//Station 3 - SMAC Homing Time Out
GVL_MASTER.stAlarms[3].aEventTimers[80]
(IN := (S_Master_SMAC.eState = E_SmacState.HOMING),PT:= T#30S );
IF GVL_MASTER.stAlarms[3].aEventTimers[80].Q  THEN 
	GVL_MASTER.stAlarms[3].aEventFlags[80] := TRUE;
END_IF
//Station 3 - SMAC Linear Homing fail
GVL_MASTER.stAlarms[3].aEventTimers[81]
(IN := (S_Master_SMAC.eState = E_SmacState.HOMING) AND stSmacIO.inStatusWordLinear.7 ,PT:= T#20S );
IF GVL_MASTER.stAlarms[3].aEventTimers[81].Q THEN 
	stAlarms[3].aEventFlags[81] := TRUE;
END_IF
//Station 3 - SMAC Linear Phasing fail
GVL_MASTER.stAlarms[3].aEventTimers[82]
(IN := (S_Master_SMAC.eState = E_SmacState.HOMING) AND stSmacIO.inStatusWordLinear.9 ,PT:= T#20S );
IF GVL_MASTER.stAlarms[3].aEventTimers[82].Q THEN
	stAlarms[3].aEventFlags[82] := TRUE;
END_IF
//Station 3 - SMAC Rotative Homing fail
GVL_MASTER.stAlarms[3].aEventTimers[83]
(IN := (S_Master_SMAC.eState = E_SmacState.HOMING) AND stSmacIO.inStatusWordRotative.7 ,PT:= T#20S );
IF GVL_MASTER.stAlarms[3].aEventTimers[83].Q THEN 
	stAlarms[3].aEventFlags[83] := TRUE;
END_IF
//Station 3 - SMAC Rotative Phasing fail
GVL_MASTER.stAlarms[3].aEventTimers[84]
(IN := (S_Master_SMAC.eState = E_SmacState.HOMING) AND stSmacIO.inStatusWordRotative.9 ,PT:= T#20S );
IF GVL_MASTER.stAlarms[3].aEventTimers[84].Q THEN 
	stAlarms[3].aEventFlags[84] := TRUE;
END_IF
END_ACTION

METHOD SetEventTexts : BOOL
VAR_INPUT
END_VAR
//Immediate Faults
GVL_MASTER.stAlarms[3].aEventTexts[1] := 'Station 3 - SMAC Linear General Fault';
GVL_MASTER.stAlarms[3].aEventTexts[2] := 'Station 3 - SMAC Linear Servo error';
GVL_MASTER.stAlarms[3].aEventTexts[3] := 'Station 3 - SMAC Rotative General Fault';
GVL_MASTER.stAlarms[3].aEventTexts[4] := 'Station 3 - SMAC Rotative Servo error';
GVL_MASTER.stAlarms[3].aEventTexts[5] := 'Station 3 - SMAC STO Fault';
GVL_MASTER.stAlarms[3].aEventTexts[6] := 'Station 3 - SMAC I2T Fault';
GVL_MASTER.stAlarms[3].aEventTexts[7] := 'Station 3 - SMAC Over temperature Fault';
GVL_MASTER.stAlarms[3].aEventTexts[8] := '';
GVL_MASTER.stAlarms[3].aEventTexts[9] := ''; 
GVL_MASTER.stAlarms[3].aEventTexts[10] := ''; 
GVL_MASTER.stAlarms[3].aEventTexts[11] := '';
GVL_MASTER.stAlarms[3].aEventTexts[12] := '';
GVL_MASTER.stAlarms[3].aEventTexts[13] := '';
GVL_MASTER.stAlarms[3].aEventTexts[14] := '';
GVL_MASTER.stAlarms[3].aEventTexts[15] := '';
GVL_MASTER.stAlarms[3].aEventTexts[16] := '';
GVL_MASTER.stAlarms[3].aEventTexts[17] := '';
GVL_MASTER.stAlarms[3].aEventTexts[18] := '';
GVL_MASTER.stAlarms[3].aEventTexts[19] := '';
GVL_MASTER.stAlarms[3].aEventTexts[20] := '';
GVL_MASTER.stAlarms[3].aEventTexts[21] := '';
GVL_MASTER.stAlarms[3].aEventTexts[22] := '';
GVL_MASTER.stAlarms[3].aEventTexts[28] := '';
GVL_MASTER.stAlarms[3].aEventTexts[29] := '';
GVL_MASTER.stAlarms[3].aEventTexts[30] := '';

//Cycle Stop Requests

GVL_MASTER.stAlarms[3].aEventTexts[80] := 'Station 3 - SMAC Homing Time Out';
GVL_MASTER.stAlarms[3].aEventTexts[81] := 'Station 3 - SMAC Linear Homing fail';
GVL_MASTER.stAlarms[3].aEventTexts[82] := 'Station 3 - SMAC Linear Phasing fail';
GVL_MASTER.stAlarms[3].aEventTexts[84] := 'Station 3 - SMAC Rotative Homing fail';
GVL_MASTER.stAlarms[3].aEventTexts[85] := 'Station 3 - SMAC Rotative Phasing fail';
GVL_MASTER.stAlarms[3].aEventTexts[86] := '';
GVL_MASTER.stAlarms[3].aEventTexts[87] := ''; 
GVL_MASTER.stAlarms[3].aEventTexts[88] := '';
GVL_MASTER.stAlarms[3].aEventTexts[89] := '';
END_METHOD

END_PROGRAM

// ---- POUs/00_MASTER/B_Safety.TcPOU
PROGRAM B_Safety
VAR


	bFirstRun						:BOOL:=TRUE;
	tonDelaySafetyRun				:Tc2_Standard.TON;
	
	
	bFirstSafetyErrorAck 			:BOOL;
	bSafetyErrorAck					:BOOL;	
	rTriggSafetyErrorAck  			:Tc2_Standard.R_TRIG;	
	tonDelayErrorAck				:Tc2_Standard.TON;
	tonSafetyErrorAckPulse			:Tc2_Standard.TON;


//-----------------------------------------------------oldschoo1
	
END_VAR

// Call for Actions:
a_Run_And_ErrorAck();
b_Cmd_SafetyDevices();
//----------------------oldschoo1

ACTION a_Run_And_ErrorAck:
// Run Safety PLC && ErrorAck: --------------------------------------------*
(**************************************************************************)


// Delay RUN on PowerUP
tonDelaySafetyRun(IN:=bFirstRun, 
				  PT:=tSystemPowerUP_Time);

IF tonDelaySafetyRun.Q 
	THEN
		GVL_MASTER.stSafety.bRunSafety 		:= TRUE;	
		bFirstRun 							:= FALSE;
		bFirstSafetyErrorAck 				:= TRUE;
END_IF

// Delay ErrorAck
tonDelayErrorAck(IN:=bFirstSafetyErrorAck, 
				 PT:=T#500MS);


// Trigger ErrorAck: ------------------------------------------------------*
rTriggSafetyErrorAck(CLK:=tonDelayErrorAck.Q OR 
						  bResetButtonRisingEdge);

IF rTriggSafetyErrorAck.Q 
	THEN
		bFirstSafetyErrorAck 	:= FALSE;
		bSafetyErrorAck 		:= TRUE;
END_IF


// Send Pulse for ErrorAck: -----------------------------------------------*
tonSafetyErrorAckPulse(IN:=bSafetyErrorAck, PT:=T#500MS);

IF bSafetyErrorAck 
							THEN
								GVL_MASTER.stSafety.bAckSafetyError := TRUE;
END_IF

IF tonSafetyErrorAckPulse.Q 
							THEN
								GVL_MASTER.stSafety.bAckSafetyError := FALSE;
								bSafetyErrorAck 					:= FALSE;
END_IF


//------------------------------------------------------------------oldschoo1
END_ACTION

ACTION b_Cmd_SafetyDevices:
// atm dev && test only 
	// map to:  stMachineStatus.bAutoCycle;  when done with dev/testing
	// map to:  stMachineStatus.bAutoCycle AND NOT stMachineStatus.bProcessCycle; //to allow operator to insert/take out the Pack fixture
  // map to:  stMachineStatus.bAutoCycle;  when done with dev/testing
IF stMachineStatus.bProcessCycle AND NOT Y_Master_Y_Axis.refY_Axis.Status.Moving THEN
	stSafety.bLightBeam_MuteCMD 	:= FALSE;
ELSE stSafety.bLightBeam_MuteCMD 	:= TRUE;
END_IF
	//stSafety.bLightBeam_MuteCMD 	:= TRUE;

IF stMachineStatus.bAutoCycle THEN
	stSafety.bTwoHands_MonitorCMD 	:= TRUE;
	stSafety.bLockDoor_CMD 			:= TRUE;
ELSE stSafety.bTwoHands_MonitorCMD 	:= FALSE;
	stSafety.bLockDoor_CMD 			:= FALSE;
END_IF
END_ACTION

ACTION z_HardwareHealth:
//to be finnished

(*
   	// TERMINAL 1 _ EK1100 - EtherCAT Coupler

	nEK1100State							AT %I*			:	UINT;	// Terminal INFO Data	
	sEK1100Status											:	STRING(200);
	

	// TERMINAL 2 _ EL6070-0033	- License Key Terminal for TC3
	
	nEL6070State							AT %I*			:	UINT;	// Terminal INFO Data	
	sEL6070Status											:	STRING(200);


	// TERMINAL 3 _ EL6910 - Safety PLC - Virtual Channels
	

	nEL6910State							AT %I*			:	UINT;	// Terminal INFO Data	
	sEL6910Status											:	STRING(200);


	// TERMINAL 4 _ EL1918 - 8 Channel Digital Safety Inputs
	

	nEL1918_1State							AT %I*			:	UINT;	// Terminal INFO Data	
	sEL1918Status											:	STRING(200);
	

	// TERMINAL 5 _ EL1918 - 8 Channel Digital Safety Inputs
                     	
	nEL1918_2State							AT %I*			:	UINT;	// Terminal INFO Data	
	sEL1918_2Status											:	STRING(200);
	

	// TERMINAL 6 _ ELEL2904 - 4 Channel Digital Safety Outputs


	nEL2904_1State							AT %I*			:	UINT;	// Terminal INFO Data	
	sEL2904_1Status											:	STRING(200);
	

	// TERMINAL 7 _ ELEL2904 - 4 Channel Digital Safety Outputs

		//Status* 
	nEL2904_2State							AT %I*			:	UINT;	// Terminal INFO Data	
	sEL2904_2Status											:	STRING(200);


	// TERMINAL 8 _ EL1809 - 16 Channel Digital Input Terminal
	
		//Status*	
	nEL1809_1State							AT %I*			:	UINT;	// Terminal INFO Data	
	sEL1809_1Status											:	STRING(200);
	
	iPSU_1_OK								AT %I*	 		: 	BOOL;	// Channel 03 - Power Supply Unit 1 OK
	iPSU_2_OK								AT %I*	 		: 	BOOL;	// Channel 04 - Power Supply Unit 2 OK
	iPSU_3_OK								AT %I*	 		: 	BOOL;	// Channel 05 - Power Supply Unit 3 OK	
	
	

	// TERMINAL 9 _ EL1809 - 16 Channel Digital Input Terminal

	nEL1809_2State							AT %I*			:	UINT;	// Terminal INFO Data
	sEL1809_2Status											:	STRING(200);
	
	// TERMINAL 10 _ EL2809	- 16 Channel Digital Output Terminal
	

	nEL2809State							AT %I*			:	UINT;	// Terminal INFO Data
	sEL2809Status											:	STRING(200);


	// TERMINAL 11 _ EL9576 - Brake Chopper Terminal

	nEL9576State							AT %I*			:	UINT;	// Terminal INFO Data
	sEL9576Status											:	STRING(200);
	

	// TERMINAL 12 _ EL7211-0010 - Servo Motor Drive

	nEL7211State							AT %I*			:	UINT;	// Terminal INFO Data
	sEL7211Status											:	STRING(200);	


	// BOX 13 _ maXYnos - Drive and Force Sensor

	nKistlermaXYmosState				   AT %I*		   :	UINT;	// Terminal INFO Data
	sKistlermaXYmosStatus								   :	STRING(200);	
	
	//--------------------------------------------------------------------------------------------------------------------------oldschoo1
*)
END_ACTION

END_PROGRAM

// ---- POUs/00_MASTER/C_Machine_CTRL.TcPOU
PROGRAM C_Machine_CTRL
VAR
	
	bFirstRun					:BOOL;
	bFirstAutoCycle				:BOOL;
	bSmacDone					:BOOL;
	bKistlerDone				:BOOL;
	rSmacDone					:R_TRIG;
	rKistlerDone				:R_TRIG;
	bStatisticsFlag				:ARRAY[0..1] OF BOOL;
	
	eMachineState				:E_MachineState:=E_MachineState.SYSTEM_POWER_UP;

	//Timers && Triggers
	tonSys_Init					:Tc2_Standard.TON:=(PT:=T#1S);
	tonSys_InitTimeout			:Tc2_Standard.TON:=(PT:=T#3M);					
	tonWAIT_SMAC_KISLR			:Tc2_Standard.TON;
	tonFirstAutoCycle			:Tc2_Standard.TON:=(PT:=T#500MS);
	
	//Process Cycle
	eCycleState					:E_ProcessCycle;
	stTotalReport				:ST_ProcessReport;
	bStartConditions			:BOOL;	
	tonTwoHandsTouching			:Tc2_Standard.TON;         
	bScrewPresent				: BOOL;
	bReservoirPresent			: BOOL;
	tonGrippersOpennedSignal	: TON;
	tonDelayExe					:Tc2_Standard.TON:=(PT:=T#100MS);
	rtrigResetModule			:Tc2_Standard.R_TRIG;
	rtrigProcessLogShift		:Tc2_Standard.R_TRIG;
	
	
	//Index
	idx							:INT;
	
END_VAR
//----------------------------------------------------------------------------oldschoo1

// Call for Actions

   b_Machine_Status();		//State machina 
	 c_ProcessCycle();	   //Master sequencer


//----------------------------------------------------------------*


// Process Report circular buffer
rtrigProcessLogShift(CLK:=eCycleState=E_ProcessCycle.Saving_DATA);

IF rtrigProcessLogShift.Q THEN 
	FOR idx:= 250 TO 2 BY -1 DO
		GVL_PERSISTENT.stProccessReportLog[idx]:=GVL_PERSISTENT.stProccessReportLog[idx-1];
	END_FOR
	GVL_PERSISTENT.stProccessReportLog[1]:=stTotalReport;
END_IF//																										||
//--------------------------------------------------------------------------------------------------------oldschoo1

ACTION b_Machine_Status:




//Timers && Triggers
tonSys_Init(IN:=stMachineStatus.bInitialising);
tonSys_InitTimeout(IN:=stMachineStatus.bInitialising);
IF stMachineStatus.eMachineState <> E_MachineState.SYSTEM_AUTO_CYCLE THEN
	bFirstAutoCycle							:= FALSE;
END_IF

//Transition IF Cycle Stop Fault OR Imediate Fault
IF NOT stMasterCtrl.bNoMachineImmediateFault THEN		
				stMachineStatus.eMachineState := E_MachineState.IMMEDIATE_FAULT;
	
ELSIF NOT stMasterCtrl.bNoCycleStopFault AND NOT stMachineStatus.bImmediateStopped THEN
				stMachineStatus.eMachineState := E_MachineState.CYCLE_STOP_FAULT;
END_IF

IF NOT GVL_Master.stMasterCTRL.bManualModeRequest THEN
	CMD_Axis.bManualMode	:=FALSE;
	CMD_Smac.bManualMode	:=FALSE;
	CMD_Kistler.bManualMode	:=FALSE;
END_IF
(****************************************************MACHINE_CTRL*******************************************************************)
//STATE MACHINE: ------------------------------------------------------------------------------------------------------------------SM
CASE stMachineStatus.eMachineState OF

E_MachineState.SYSTEM_POWER_UP: 		// ------------------------------------------------------------------------------POWER_UP

				IF tonSystemPowerUP.Q THEN
						stMachineStatus.eMachineState := E_MachineState.IMMEDIATE_STOPPED;//
				END_IF
	
E_MachineState.IMMEDIATE_STOPPED:		// ---------------------------------------------------------------------IMMEDIATE_STOPPED

				IF stMasterCtrl.bNoMachineImmediateFault AND bResetButtonFallingEdge THEN
						stMachineStatus.eMachineState := E_MachineState.SYSTEM_INITIALISING;//
						
				ELSIF NOT stMasterCtrl.bNoCycleStopFault THEN
						stMachineStatus.eMachineState := E_MachineState.CYCLE_STOP_FAULT;//
					
				ELSIF NOT stMasterCtrl.bNoMachineImmediateFault THEN
					stMachineStatus.eMachineState := E_MachineState.IMMEDIATE_FAULT;//	
				END_IF		


E_MachineState.SYSTEM_INITIALISING:		// -------------------------------------------------------------------SYSTEM_INITIALISING		

				IF tonSys_Init.Q THEN
						CMD_Axis.bEnable	:=TRUE;
						CMD_Smac.bEnable	:=TRUE;
						CMD_Kistler.bEnable	:=TRUE;
						
						CMD_Axis.bAbort		:=FALSE;
						CMD_Smac.bAbort		:=FALSE;
						CMD_Kistler.bAbort	:=FALSE;
				END_IF

				//IF Axis_STATUS.bReady AND Kistler_STATUS.bReady  AND Smac_STATUS.bReady THEN 
				 IF Axis_STATUS.bReady AND Kistler_STATUS.bReady AND ( GVL_PERSISTENT.bSMACEnable AND Smac_STATUS.bReady OR NOT GVL_PERSISTENT.bSMACEnable) THEN //**LAA  29092025
										stMachineStatus.eMachineState:= E_MachineState.SYSTEM_READY_TO_START;//
				END_IF

				IF bStopButtonFallingEdge OR 
			 	  (stMasterCtrl.bNoMachineImmediateFault AND 
			 	  (stMasterCtrl.bCycleStopRequest OR tonSys_InitTimeout.Q) AND 
			       stMasterCtrl.bAllActionsStopped)
					THEN
										stMachineStatus.eMachineState := E_MachineState.CYCLE_STOPPED;//
						
				ELSIF stMasterCtrl.bNoMachineImmediateFault AND NOT stMasterCtrl.bNoCycleStopFault 
					THEN		
										stMachineStatus.eMachineState := E_MachineState.CYCLE_STOP_FAULT;//
			
				ELSIF NOT stMasterCtrl.bNoMachineImmediateFault 
					THEN
										stMachineStatus.eMachineState := E_MachineState.IMMEDIATE_FAULT;//
				END_IF
			
					
E_MachineState.SYSTEM_READY_TO_START:	// -------------------------------------------------------------------SYSTEM_READY_TO_START<<<

				IF 	 bStartButtonFallingEdge AND stMasterCtrl.bAllModulesReady THEN
					
										stMachineStatus.eMachineState := E_MachineState.SYSTEM_AUTO_CYCLE;//
				
				ELSIF bStopButtonFallingEdge THEN
					
										stMachineStatus.eMachineState := E_MachineState.STOPPING;//
										
				ELSIF stMasterCtrl.bNoMachineImmediateFault AND NOT stMasterCtrl.bNoCycleStopFault THEN	
	
										stMachineStatus.eMachineState := E_MachineState.CYCLE_STOP_FAULT;//
			
				ELSIF NOT stMasterCtrl.bNoMachineImmediateFault THEN
										stMachineStatus.eMachineState := E_MachineState.IMMEDIATE_FAULT;//
				ELSIF GVL_Master.stMasterCTRL.bManualModeRequest AND stMasterCtrl.bNoMachineImmediateFault AND stMasterCtrl.bNoCycleStopFault THEN
										stMachineStatus.eMachineState := E_MachineState.MANUAL_MODE;//
				END_IF

				

E_MachineState.SYSTEM_AUTO_CYCLE:		// ---------------------------------------------------------------------SYSTEM_AUTO_CYCLE	

				IF bStopButtonFallingEdge THEN					
										stMachineStatus.eMachineState := E_MachineState.STOPPING;//
						
				ELSIF stMasterCtrl.bCycleStopRequest THEN 
					
										stMachineStatus.eMachineState := E_MachineState.STOPPING;//
										
				ELSIF stMasterCtrl.bNoMachineImmediateFault AND NOT stMasterCtrl.bNoCycleStopFault THEN	
	
										stMachineStatus.eMachineState := E_MachineState.CYCLE_STOP_FAULT;//
			
				ELSIF NOT stMasterCtrl.bNoMachineImmediateFault THEN
										stMachineStatus.eMachineState := E_MachineState.IMMEDIATE_FAULT;//
				END_IF	

E_MachineState.SYSTEM_STANDBY:;//



E_MachineState.STOPPING:				// ------------------------------------------------------------------------------STOPPING

				IF stMasterCtrl.bAllActionsStopped THEN
										stMachineStatus.eMachineState := E_MachineState.CYCLE_STOPPED;//					
				END_IF
				CMD_Axis.bEnable	:=FALSE;
				CMD_Smac.bEnable	:=FALSE;
				CMD_Kistler.bEnable	:=FALSE;
				
				CMD_Axis.bAbort		:=TRUE;
				CMD_Smac.bAbort		:=TRUE;
				CMD_Kistler.bAbort	:=TRUE;

E_MachineState.CYCLE_STOPPED:			// -------------------------------------------------------------------------CYCLE_STOPPED

				IF stMasterCtrl.bNoCycleStopFault   AND 
	      		NOT stMasterCtrl.bCycleStopRequest  AND 
                               bResetButtonFallingEdge

									THEN	
										stMachineStatus.eMachineState := E_MachineState.SYSTEM_INITIALISING;		
				END_IF	

E_MachineState.IMMEDIATE_FAULT:			// -----------------------------------------------------------------------IMMEDIATE_FAULT
				
				CMD_Axis.bEnable	:=FALSE;
				CMD_Smac.bEnable	:=FALSE;
				CMD_Kistler.bEnable	:=FALSE;
						
				CMD_Axis.bAbort		:=TRUE;
				CMD_Smac.bAbort		:=TRUE;
				CMD_Kistler.bAbort	:=TRUE;
				
				IF stMasterCtrl.bNoMachineImmediateFault	THEN
										stMachineStatus.eMachineState := E_MachineState.IMMEDIATE_STOPPED;		
				END_IF

E_MachineState.CYCLE_STOP_FAULT:		// ----------------------------------------------------------------------CYCLE_STOP_FAULT

				CMD_Axis.bEnable	:=FALSE;
				CMD_Smac.bEnable	:=FALSE;
				CMD_Kistler.bEnable	:=FALSE;
						
				CMD_Axis.bAbort		:=TRUE;
				CMD_Smac.bAbort		:=TRUE;
				CMD_Kistler.bAbort	:=TRUE;
				
				IF stMasterCtrl.bNoCycleStopFault THEN
										stMachineStatus.eMachineState := E_MachineState.CYCLE_STOPPED;
				END_IF	


E_MachineState.MANUAL_MODE:;//

				IF bStopButtonFallingEdge OR NOT GVL_Master.stMasterCTRL.bManualModeRequest THEN
					
										stMachineStatus.eMachineState := E_MachineState.STOPPING;//
										
										CMD_Axis.bManualMode:=FALSE;
										CMD_Smac.bManualMode:=FALSE;
										CMD_Kistler.bManualMode:=FALSE;
										CMD_Axis.bAbort		:=TRUE;
										CMD_Smac.bAbort		:=TRUE;
										CMD_Kistler.bAbort	:=TRUE;
				ELSIF stMasterCtrl.bNoMachineImmediateFault AND NOT stMasterCtrl.bNoCycleStopFault THEN	
	
										stMachineStatus.eMachineState := E_MachineState.CYCLE_STOP_FAULT;//
										
										CMD_Axis.bManualMode:=FALSE;
										CMD_Smac.bManualMode:=FALSE;
										CMD_Kistler.bManualMode:=FALSE;
										CMD_Axis.bAbort		:=TRUE;
										CMD_Smac.bAbort		:=TRUE;
										CMD_Kistler.bAbort	:=TRUE;
			
				ELSIF NOT stMasterCtrl.bNoMachineImmediateFault THEN
							
										stMachineStatus.eMachineState := E_MachineState.IMMEDIATE_FAULT;//
				
										CMD_Axis.bManualMode:=FALSE;
										CMD_Smac.bManualMode:=FALSE;
										CMD_Kistler.bManualMode:=FALSE;
										CMD_Axis.bAbort		:=TRUE;
										CMD_Smac.bAbort		:=TRUE;
										CMD_Kistler.bAbort	:=TRUE;
										
				ELSE 					CMD_Axis.bManualMode:=TRUE;
										CMD_Smac.bManualMode:=TRUE;
										CMD_Kistler.bManualMode:=TRUE;
				END_IF
ELSE
stMachineStatus.eMachineState:=E_MachineState.SYSTEM_POWER_UP;		
END_CASE									// ------------------------------------------------------------------------------- END SM


(******************************************************MACHINE_STATUS***************************************************************)
// Status Flags -----------------------------------------------------------------------------------------------------STATUS_FLAGS
stMachineStatus.bSystemPowerUp 			:= (stMachineStatus.eMachineState = E_MachineState.SYSTEM_POWER_UP);
stMachineStatus.bImmediateStopped 		:= (stMachineStatus.eMachineState = E_MachineState.IMMEDIATE_STOPPED);
stMachineStatus.bInitialising 			:= (stMachineStatus.eMachineState = E_MachineState.SYSTEM_INITIALISING);
stMachineStatus.bReadyToStart 			:= (stMachineStatus.eMachineState = E_MachineState.SYSTEM_READY_TO_START);
stMachineStatus.bAutoCycle 				:= (stMachineStatus.eMachineState = E_MachineState.SYSTEM_AUTO_CYCLE);
stMachineStatus.bStandby 				:= (stMachineStatus.eMachineState = E_MachineState.SYSTEM_STANDBY);
stMachineStatus.bStopping 				:= (stMachineStatus.eMachineState = E_MachineState.STOPPING);
stMachineStatus.bCycleStopped 			:= (stMachineStatus.eMachineState = E_MachineState.CYCLE_STOPPED);
stMachineStatus.bImmediateFault 		:= (stMachineStatus.eMachineState = E_MachineState.IMMEDIATE_FAULT);
stMachineStatus.bCycleStopFault 		:= (stMachineStatus.eMachineState = E_MachineState.CYCLE_STOP_FAULT);
stMachineStatus.bManualMode 			:= (stMachineStatus.eMachineState = E_MachineState.MANUAL_MODE);

//Transition Flags -----------------------------------------------------------------------------------------------TRANZITION_FLAGS
stMasterCtrl.bAllActionsStopped			:= (Axis_STATUS.bReady AND Kistler_STATUS.bReady AND ( GVL_PERSISTENT.bSMACEnable AND Smac_STATUS.bReady OR NOT GVL_PERSISTENT.bSMACEnable) ) OR  //**LAA 29092025
										   (NOT Axis_STATUS.bBusy AND NOT Kistler_STATUS.bBusy );
										   
stMasterCtrl.bAllModulesReady			:= (Axis_STATUS.bReady AND Kistler_STATUS.bReady AND ( GVL_PERSISTENT.bSMACEnable AND Smac_STATUS.bReady OR NOT GVL_PERSISTENT.bSMACEnable)); //**LAA 29092025

(*stMasterCtrl.bAllActionsStopped			:= (Axis_STATUS.bReady AND Kistler_STATUS.bReady AND Smac_STATUS.bReady ) OR
										   (NOT Axis_STATUS.bBusy AND NOT Kistler_STATUS.bBusy );
										   
stMasterCtrl.bAllModulesReady			:= (Axis_STATUS.bReady AND Kistler_STATUS.bReady AND Smac_STATUS.bReady ); 

*)
END_ACTION

ACTION c_ProcessCycle:
//Timers
tonDelayExe(IN:=(eCycleState=E_ProcessCycle.AXIS_HOME AND Axis_STATUS.bReady) OR
				(eCycleState=E_ProcessCycle.AXIS_CMD_1 AND Axis_STATUS.bReady) OR
				(eCycleState=E_ProcessCycle.AXIS_CMD_2 AND Axis_STATUS.bReady) OR
				(eCycleState=E_ProcessCycle.AXIS_CMD_3 AND Axis_STATUS.bReady) OR
				(eCycleState=E_ProcessCycle.SMAC_CMD_1 AND Smac_STATUS.bReady) OR
				((eCycleState=E_ProcessCycle.CMD_SMAC_KISLR OR eCycleState=E_ProcessCycle.CMD_KISLR )AND (CMD_Kistler.bExecute OR NOT bReservoir_Present)AND (GVL_PERSISTENT.bSMACEnable AND CMD_Smac.bExecute OR NOT bScrewPresent ))
);  //AND Smac_STATUS.bReady));				//to finish
				
tonGrippersOpennedSignal( IN :=  NOT stSmac.bGripperA_ClosedSensor AND NOT stSmac.bGripperA_ClosedSensor, PT := T#1S);
tonWAIT_SMAC_KISLR(IN := eCycleState = E_ProcessCycle.WAIT_SMAC_KISLR,PT := T#500MS);
tonFirstAutoCycle( IN := eCycleState = E_ProcessCycle.IDLE AND stMachineStatus.bAutoCycle);
(******************************************************START CONDITIONS******************************************************)				
// Start Conditions: 
// - Optional add HMI PopUp if Pack fixture is in but NOT all 3 parts present -	
		
tonTwoHandsTouching(IN:=stSafety.bTwoHands_Signal, PT:=T#500MS);       // **LAA 03/12/2025 > it was too slow PT:=T#2S);

bStartConditions 		 := (tonTwoHandsTouching.Q AND 
							stMachineStatus.bAutoCycle AND
							GVL_MASTER.bPuck_Present);
							//AND bGearBox_Present 
					
							
//Reset Module --------------------------------------------------------------------------------------------------------------*
IF bResetButtonRisingEdge OR 
stMachineStatus.bCycleStopFault OR stMachineStatus.bImmediateFault OR stMachineStatus.bImmediateStopped
THEN eCycleState:=E_ProcessCycle.RESET_ALL_CMD;END_IF
//KISTLER / SMAC DONE---------------------------------------------------------------------------------------------------------*
rSmacDone( CLK := Smac_STATUS.bDone );					
rKistlerDone( CLK := Kistler_STATUS.bDone );					

IF rKistlerDone.Q THEN 
	bKistlerDone		:= TRUE;
END_IF
IF rSmacDone.Q THEN
	bSmacDone			:= TRUE;
END_IF

(************************************************************CTRL*************************************************************)
//STATE MACHINE: -----------------------------------------------------------------------------------------------------------SM
CASE eCycleState OF
						(****************************************************************IDLE********************************)
E_ProcessCycle.IDLE:	//-----------------------------------------------------------------------------------------------IDLE
									IF bStartConditions AND GVL_PERSISTENT.bSMACEnable THEN   //**LAA 29092025
										eCycleState:=E_ProcessCycle.AXIS_CMD_1;
										stTotalReport.bKis_Pass								:= FALSE;
										stTotalReport.bKis_Fail								:= FALSE;
										stTotalReport.bSmac_Pass							:= FALSE;
										stTotalReport.bSmac_Fail							:= FALSE;
										GVL_IO.qCycleIndicator_RedLED						:= FALSE;
										GVL_IO.qCycleIndicator_GreenLED						:= FALSE;
										S_Master_SMAC.bCloseGripper							:= FALSE;
										ELSIF bStartConditions AND NOT GVL_PERSISTENT.bSMACEnable THEN // *LAA  29092025
											eCycleState:=E_ProcessCycle.AXIS_CMD_2;
											stTotalReport.bKis_Pass								:= FALSE;
											stTotalReport.bKis_Fail								:= FALSE;
											stTotalReport.bSmac_Pass							:= FALSE;
											stTotalReport.bSmac_Fail							:= FALSE;
											GVL_IO.qCycleIndicator_RedLED						:= FALSE;
											GVL_IO.qCycleIndicator_GreenLED						:= FALSE;
											S_Master_SMAC.bCloseGripper							:= FALSE;
									END_IF
									 IF NOT bFirstAutoCycle AND GVL_MASTER.bPuck_Present AND
										NOT tonFirstAutoCycle.Q AND stMachineStatus.bAutoCycle THEN
										eCycleState:=E_ProcessCycle.AXIS_CMD_3;
										stTotalReport.bKis_Pass								:= FALSE;
										stTotalReport.bKis_Fail								:= FALSE;
										stTotalReport.bSmac_Pass							:= FALSE;
										stTotalReport.bSmac_Fail							:= FALSE;
										GVL_IO.qCycleIndicator_RedLED						:= FALSE;
										GVL_IO.qCycleIndicator_GreenLED						:= FALSE;
										S_Master_SMAC.bCloseGripper							:= FALSE;
									END_IF
									//Just Idleing like chilling here
									CMD_Smac.bFixtureGripper		:= FALSE;
									CMD_Smac.bGuideGripper			:= FALSE;
									IF stMachineStatus.bAutoCycle AND NOT GVL_MASTER.bPuck_Present THEN
										GVL_HMI.sMessageToOperator	:='Insert Nest';
									ELSIF stMachineStatus.bAutoCycle AND GVL_MASTER.bPuck_Present THEN
										GVL_HMI.sMessageToOperator	:='Put two hands to start Cycle Process';
									ELSIF NOT stMachineStatus.bAutoCycle AND  stMachineStatus.bReadyToStart THEN
									GVL_HMI.sMessageToOperator	:='Press START to Begin';
									ELSIF NOT stMachineStatus.bAutoCycle AND  NOT stMachineStatus.bReadyToStart THEN
									GVL_HMI.sMessageToOperator	:='Press RESET';
									END_IF
									
							(************************************************************CYCLE******************************)									
E_ProcessCycle.AXIS_CMD_1:	//-------------------------------------------------------------------------------------AXIS_CMD_1

									IF Axis_STATUS.bReady THEN
											stY_Axis.bSetToPosition[1]	:=TRUE;
									END_IF

									IF tonDelayExe.Q THEN
											CMD_Axis.bExecute			:=TRUE;
											eCycleState:=E_ProcessCycle.WAIT_AXIS_CMD_1;
									END_IF
									GVL_HMI.sMessageToOperator	:='Axis Y Moving to Position 1';
									bFirstAutoCycle						:=TRUE;
									
	
E_ProcessCycle.WAIT_AXIS_CMD_1:	//----------------------------------------------------------------------------WAIT_AXIS_CMD_1
							 		IF GVL_PERSISTENT.bSMACEnable AND Axis_STATUS.bDone AND bScrew_Present THEN
											stY_Axis.bSetToPosition[1]	:=FALSE;
											CMD_Axis.bExecute			:=FALSE;
											bScrewPresent				:=TRUE;
											eCycleState:=E_ProcessCycle.SMAC_CMD_1;
									ELSIF  GVL_PERSISTENT.bSMACEnable AND Axis_STATUS.bDone AND NOT bScrew_Present OR NOT GVL_PERSISTENT.bSMACEnable THEN
											stY_Axis.bSetToPosition[1]	:=FALSE;
											CMD_Axis.bExecute			:=FALSE;
											bScrewPresent				:=FALSE;
											eCycleState:=E_ProcessCycle.AXIS_CMD_2;
									END_IF
									
									
E_ProcessCycle.SMAC_CMD_1:	//-------------------------------------------------------------------------------------SMAC_CMD_1		//to finish
									IF  Smac_STATUS.bReady THEN
										stSmac.bSet_PickScrew				:=TRUE;
										CMD_Smac.bExecute					:=TRUE;
									END_IF
									IF  Smac_Status.bBusy THEN
										eCycleState:=E_ProcessCycle.WAIT_SMAC_CMD_1;
									END_IF
									
									GVL_HMI.sMessageToOperator	:='Smac Picking Screw Part';

	
E_ProcessCycle.WAIT_SMAC_CMD_1:	//----------------------------------------------------------------------------WAIT_SMAC_CMD_1		//to finish
									//Wait for Smac device to feedback 
									IF Smac_STATUS.bFirstPartOfCycleDone THEN
										eCycleState:=E_ProcessCycle.AXIS_CMD_2;	
										CMD_Smac.bExecute				:=FALSE;
									END_IF

E_ProcessCycle.AXIS_CMD_2:	//-------------------------------------------------------------------------------------AXIS_CMD_2
							 		
											stY_Axis.bSetToPosition[2]	:=TRUE;
									

									IF tonDelayExe.Q AND Axis_STATUS.bReady THEN
											CMD_Axis.bExecute			:=TRUE;
											eCycleState:=E_ProcessCycle.WAIT_AXIS_CMD_2;
									END_IF	
									
									GVL_HMI.sMessageToOperator	:='Axis Y Moving to Position 2';

E_ProcessCycle.WAIT_AXIS_CMD_2:	//----------------------------------------------------------------------------WAIT_AXIS_CMD_2
						 		IF Axis_STATUS.bDone  AND GVL_PERSISTENT.bSMACEnable THEN
											stY_Axis.bSetToPosition[2]	:=FALSE;
											CMD_Axis.bExecute			:=FALSE;
											eCycleState:=E_ProcessCycle.GRIPPERS_CMD_1;
											ELSIF Axis_STATUS.bDone AND NOT GVL_PERSISTENT.bSMACEnable THEN 
												stY_Axis.bSetToPosition[2]	:=FALSE;
												CMD_Axis.bExecute			:=FALSE;
												eCycleState:=E_ProcessCycle.CMD_KISLR;;
									END_IF	
E_ProcessCycle.GRIPPERS_CMD_1: //------------------------------------------------------------------------------GRIPPERS_CMD_1
								
									CMD_Smac.bFixtureGripper		:= TRUE;
									CMD_Smac.bGuideGripper			:= TRUE;
								
								eCycleState:=E_ProcessCycle.WAIT_GRIPPERS_CMD_1;
								
								

E_ProcessCycle.WAIT_GRIPPERS_CMD_1: //--------------------------------------------------------------------WAIT_GRIPPERS_CMD_1
								IF stSmac.bGripperA_ClosedSensor AND stSmac.bGripperA_ClosedSensor AND 
									(bScrewPresent OR bPuck_Present) THEN
									eCycleState:=E_ProcessCycle.CMD_SMAC_KISLR;
								ELSIF stSmac.bGripperA_ClosedSensor AND stSmac.bGripperA_ClosedSensor AND // *LAA ????????
									(bScrewPresent OR bPuck_Present) THEN
									eCycleState:=E_ProcessCycle.STORE_PROC_DATA;
								END_IF

E_ProcessCycle.CMD_SMAC_KISLR:	//-------------------------------------------------------------------------CMD_SMAC_AND_KISLR		//to finish
							 		IF Kistler_STATUS.bReady THEN // AND Smac_STATUS.bReady
											IF bReservoir_Present THEN
												CMD_Kistler.bExecute		:=TRUE;
												bReservoirPresent			:=TRUE;
											END_IF
											IF bScrewPresent THEN
											stSmac.bSet_ScrewItIn		:=TRUE;
											CMD_Smac.bExecute			:=TRUE;
											END_IF
									END_IF

									IF tonDelayExe.Q THEN
										
											eCycleState:=E_ProcessCycle.WAIT_SMAC_KISLR;
									END_IF				
									GVL_HMI.sMessageToOperator	:='Kistler and Screw Process';

E_ProcessCycle.WAIT_SMAC_KISLR:	//----------------------------------------------------------------------------WAIT_SMAC_KISLR		//to finish
						 			IF (bKistlerDone OR NOT bReservoir_Present) AND (bSmacDone OR NOT bScrewPresent) THEN
											CMD_Kistler.bExecute		:=FALSE;
											stSmac.bSet_ScrewItIn		:=FALSE;
											CMD_Smac.bExecute			:=FALSE;
											//open guide gripper
											eCycleState:=E_ProcessCycle.STORE_PROC_DATA;
									END_IF	
//**************************************LAA******************************************************************//			

E_ProcessCycle.CMD_KISLR:	//-------------------------------------------------------------------------CMD_SMAC_AND_KISLR		//to finish
							 		IF Kistler_STATUS.bReady THEN // AND Smac_STATUS.bReady
											IF bReservoir_Present THEN
												CMD_Kistler.bExecute		:=TRUE;
												bReservoirPresent			:=TRUE;
											END_IF
									END_IF

									IF tonDelayExe.Q THEN
										
											eCycleState:=E_ProcessCycle.WAIT_KISLR;
									END_IF				
									GVL_HMI.sMessageToOperator	:='Kistler processing';

E_ProcessCycle.WAIT_KISLR:	//----------------------------------------------------------------------------WAIT_SMAC_KISLR		//to finish
						 			IF (bKistlerDone OR NOT bReservoir_Present) THEN
											CMD_Kistler.bExecute		:=FALSE;
											eCycleState:=E_ProcessCycle.STORE_PROC_DATA;
									END_IF	
//**************************************LAA******************************************************************//			
E_ProcessCycle.STORE_PROC_DATA:	//----------------------------------------------------------------------------STORE_PROC_DATA		//to finish
		
	bKistlerDone 			:= FALSE;
	bSmacDone 				:= FALSE;
	
	IF bReservoirPresent THEN
		stTotalReport.bKis_Pass								:=K_Master_Kistler.stKistlerReport.bKis_Pass;
		stTotalReport.bKis_Fail								:=K_Master_Kistler.stKistlerReport.bKis_Fail;
		stTotalReport.rKis_HighestRecordedForce				:=K_Master_Kistler.stKistlerReport.rKis_HighestRecordedForce;
		stTotalReport.rKis_LowestRecordedForce				:=K_Master_Kistler.stKistlerReport.rKis_LowestRecordedForce;
		stTotalReport.rKis_DistanceRecord					:=K_Master_Kistler.stKistlerReport.rKis_DistanceRecord;
		stTotalReport.rKis_Settings_ForceUpperTreshold		:=K_Master_Kistler.stKistlerReport.rKis_Settings_ForceUpperTreshold;
		stTotalReport.rKis_Settings_ForceLowerTreshold		:=K_Master_Kistler.stKistlerReport.rKis_Settings_ForceLowerTreshold;
		stTotalReport.rKis_Settings_StartMeasurePoint		:=K_Master_Kistler.stKistlerReport.rKis_Settings_StartMeasurePoint;
		stTotalReport.rKis_Settings_ReservoirBottomPoint	:=K_Master_Kistler.stKistlerReport.rKis_Settings_ReservoirBottomPoint;
		IF stTotalReport.bKis_Pass THEN
			stTotalReport.sKis_Result							:='PASS';
		ELSIF stTotalReport.bKis_FaiL THEN
			stTotalReport.sKis_Result							:='FAIL';
		ELSE stTotalReport.sKis_Result							:='';
		END_IF
	ELSE
		stTotalReport.bKis_Pass								:=FALSE;
		stTotalReport.bKis_Fail								:=FALSE;
		stTotalReport.rKis_HighestRecordedForce				:=0;
		stTotalReport.rKis_LowestRecordedForce				:=0;
		stTotalReport.rKis_Settings_ForceUpperTreshold		:=0;
		stTotalReport.rKis_Settings_ForceLowerTreshold		:=0;
		stTotalReport.rKis_Settings_StartMeasurePoint		:=0;
		stTotalReport.rKis_Settings_ReservoirBottomPoint	:=0;
		stTotalReport.sKis_Result							:='';
	END_IF
	IF GVL_PERSISTENT.bSMACEnable AND bScrewPresent THEN
		stTotalReport.rSmac_Settings_LinearAcc				:=S_Master_SMAC.stSmacReport.rSmac_Settings_LinearAcc;
		stTotalReport.rSmac_Settings_LinearVel				:=S_Master_SMAC.stSmacReport.rSmac_Settings_LinearVel;
		stTotalReport.rSmac_Settings_RotativeAcc			:=S_Master_SMAC.stSmacReport.rSmac_Settings_RotativeAcc;
		stTotalReport.rSmac_Settings_RotativeVel			:=S_Master_SMAC.stSmacReport.rSmac_Settings_RotativeVel;
		stTotalReport.rSmac_Settings_LinearTorque			:=S_Master_SMAC.stSmacReport.rSmac_Settings_LinearTorque;
		stTotalReport.rSmac_MaxDistanceReached				:=S_Master_SMAC.stSmacReport.rSmac_MaxDistanceReached;
		stTotalReport.bSmac_Pass							:=S_Master_SMAC.stSmacReport.bSmac_Pass;
		stTotalReport.bSmac_Fail							:=S_Master_SMAC.stSmacReport.bSmac_Fail;
		IF stTotalReport.bSmac_Pass THEN
			stTotalReport.sSmac_Result							:='PASS';
		ELSIF stTotalReport.bSmac_Fail THEN
			stTotalReport.sSmac_Result							:='FAIL';
		ELSE stTotalReport.sSmac_Result							:='';
		END_IF
	ELSE
		stTotalReport.rSmac_Settings_LinearAcc				:=0;
		stTotalReport.rSmac_Settings_LinearVel				:=0;
		stTotalReport.rSmac_Settings_RotativeAcc			:=0;
		stTotalReport.rSmac_Settings_RotativeVel			:=0;
		stTotalReport.rSmac_Settings_LinearTorque			:=0;
		stTotalReport.rSmac_MaxDistanceReached				:=0;
		stTotalReport.bSmac_Pass							:=FALSE;
		stTotalReport.bSmac_Fail							:=FALSE;
		stTotalReport.sSmac_Result							:='';
	END_IF
	
	stTotalReport.sDate										:= GVL_MASTER.sSystemDate;
	stTotalReport.sTime										:= GVL_MASTER.sSystemTime;
	
	//STATISTICS
	IF bReservoirPresent AND stTotalReport.bKis_Pass AND NOT bStatisticsFlag[0] THEN
		GVL_PERSISTENT.nKistlerGoodParts					:= GVL_PERSISTENT.nKistlerGoodParts + 1;
		GVL_PERSISTENT.nKistlerTotalGoodParts				:= GVL_PERSISTENT.nKistlerTotalGoodParts + 1;
		bStatisticsFlag[0]									:= TRUE;
	END_IF
	IF bReservoirPresent AND stTotalReport.bKis_Fail AND NOT bStatisticsFlag[0] THEN
		GVL_PERSISTENT.nKistlerBadParts						:= GVL_PERSISTENT.nKistlerBadParts + 1;
		GVL_PERSISTENT.nKistlerTotalBadParts				:= GVL_PERSISTENT.nKistlerTotalBadParts + 1;
		bStatisticsFlag[0]									:= TRUE;
	END_IF
	
	IF bScrewPresent AND stTotalReport.bSmac_Pass AND NOT bStatisticsFlag[1] THEN
		GVL_PERSISTENT.nSmacGoodParts						:= GVL_PERSISTENT.nSmacGoodParts + 1;
		GVL_PERSISTENT.nSmacTotalGoodParts					:= GVL_PERSISTENT.nSmacTotalGoodParts + 1;
		bStatisticsFlag[1]									:= TRUE;
	END_IF
		IF bScrewPresent AND stTotalReport.bSmac_Fail AND NOT bStatisticsFlag[1] THEN
		GVL_PERSISTENT.nSmacBadParts						:= GVL_PERSISTENT.nSmacBadParts + 1;
		GVL_PERSISTENT.nSmacTotalBadParts					:= GVL_PERSISTENT.nSmacTotalBadParts + 1;
		bStatisticsFlag[1]									:= TRUE;
	END_IF
	
			
			
									eCycleState:=E_ProcessCycle.Saving_DATA;	
E_ProcessCycle.Saving_DATA: //------------------------------------------------------------------------------------Saving_DATA
									eCycleState:=E_ProcessCycle.GRIPPERS_CMD_2;
									bStatisticsFlag[0]									:= FALSE;
									bStatisticsFlag[1]									:= FALSE;
									IF (bReservoirPresent AND stTotalReport.bKis_Pass) OR 
										(bScrewPresent AND stTotalReport.bSmac_Pass)THEN
										GVL_IO.qCycleIndicator_GreenLED						:= TRUE;
									ELSIF (bReservoirPresent AND stTotalReport.bKis_Fail) OR 
										(bScrewPresent AND stTotalReport.bSmac_Fail) THEN
										GVL_IO.qCycleIndicator_RedLED						:= TRUE;		
									END_IF
E_ProcessCycle.GRIPPERS_CMD_2: //------------------------------------------------------------------------------GRIPPERS_CMD_1
								
								CMD_Smac.bFixtureGripper		:= FALSE;
								CMD_Smac.bGuideGripper			:= FALSE;
								
								eCycleState:=E_ProcessCycle.WAIT_GRIPPERS_CMD_2;
								
								
								

E_ProcessCycle.WAIT_GRIPPERS_CMD_2: //--------------------------------------------------------------------WAIT_GRIPPERS_CMD_1
								IF tonGrippersOpennedSignal.Q THEN
								eCycleState:=E_ProcessCycle.AXIS_CMD_3;
								END_IF
			
E_ProcessCycle.AXIS_CMD_3:	//-------------------------------------------------------------------------------------AXIS_CMD_3
						 		IF Axis_STATUS.bReady THEN
											stY_Axis.bSetToPosition[3]	:=TRUE;
									END_IF

									IF tonDelayExe.Q THEN
											CMD_Axis.bExecute			:=TRUE;
											eCycleState:=E_ProcessCycle.WAIT_AXIS_CMD_3;
									END_IF		
								GVL_HMI.sMessageToOperator	:='Take Nest please';

E_ProcessCycle.WAIT_AXIS_CMD_3:	//----------------------------------------------------------------------------WAIT_AXIS_CMD_3
							 		IF Axis_STATUS.bDone THEN
											stY_Axis.bSetToPosition[3]	:=FALSE;
											CMD_Axis.bExecute			:=FALSE;
											eCycleState:=E_ProcessCycle.AXIS_HOME;
									END_IF


E_ProcessCycle.AXIS_HOME:	//-------------------------------------------------------------------------------------AXIS_HOME
							 		IF Axis_STATUS.bReady THEN
											stY_Axis.bSetToHome			:=TRUE;
											Y_Master_Y_Axis.bRetract 	:=TRUE;
									END_IF

									IF tonDelayExe.Q THEN
											CMD_Axis.bExecute			:=TRUE;
											eCycleState:=E_ProcessCycle.WAIT_AXIS_HOME;
									END_IF
									GVL_HMI.sMessageToOperator	:='Axis Y Homing';

E_ProcessCycle.WAIT_AXIS_HOME:	//----------------------------------------------------------------------------WAIT_AXIS_HOME
							 		IF Axis_STATUS.bDone THEN
											stY_Axis.bSetToHome			:=FALSE;
											CMD_Axis.bExecute			:=FALSE;
											Y_Master_Y_Axis.bRetract 	:=FALSE;
											eCycleState:=E_ProcessCycle.IDLE;
									END_IF
									bFirstAutoCycle						:=TRUE;

									
								(*********************************************************RESET*****************************)
E_ProcessCycle.RESET_ALL_CMD:	//------------------------------------------------------------------------------RESET_ALL_CMD

											CMD_Axis.bExecute									:=FALSE;
											CMD_Smac.bExecute									:=FALSE;
											CMD_Kistler.bExecute								:=FALSE;
											
											stSmac.bSet_PickScrew								:=FALSE;											
											stSmac.bSet_ScrewItIn								:=FALSE;
											CMD_Smac.bFixtureGripper							:= FALSE;
											CMD_Smac.bGuideGripper								:= FALSE;


											stY_Axis.bSetToHome									:=FALSE;
											Y_Master_Y_Axis.bRetract 							:=FALSE;
											stY_Axis.bSetToPosition[1]							:=FALSE;
											stY_Axis.bSetToPosition[2]							:=FALSE;
											stY_Axis.bSetToPosition[3]							:=FALSE;
											
											bKistlerDone 										:= FALSE;
											bSmacDone 											:= FALSE;
											bScrewPresent										:= FALSE;
											
											
											


											eCycleState:=E_ProcessCycle.IDLE;
											
	
ELSE
eCycleState:=E_ProcessCycle.RESET_ALL_CMD;		
END_CASE	// -------------------------------------------------------------------------------------------------------- END SM

(************************************************************STATUS************************************************************)
stMachineStatus.bProcessCycle := eCycleState <> E_ProcessCycle.IDLE AND eCycleState <> E_ProcessCycle.RESET_ALL_CMD;

//---------------------------------------------------------------------------------------------------------------------oldschoo1
END_ACTION

END_PROGRAM

// ---- POUs/02_HMI/A_HMI.TcPOU
PROGRAM A_HMI
VAR
	fbStringFormatter       :	Tc2_Utilities.FB_FormatString;
	fbScaleSmacMan			: 	FB_Scale;
	fbScaleKistlerMan		: 	FB_Scale;
	fbScaleSmacCyc			: 	FB_Scale;
	fbScaleKistlerCyc		: 	FB_Scale;
	fbScaleScrew			: 	FB_Scale;
	tonButtonPressed		: 	TON;
	
	sUserGroupID			:	STRING;
	nSize					:	UDINT					:=9;
	nLen					:	UDINT					:=18;
	npos					:	UDINT					:=1;
	tonUserLogOut			:	TON;
	tUserLoggedIn			:	TON;
	rUserLoggedIn			: 	R_TRIG;
	bUserLoggedIn			:	BOOL;
	closeChrome 			: 	NT_StartProcess;
	OpenKistlerHMI 			: 	NT_StartProcess;
	ntShutdown				: TC2_Utilities.NT_Shutdown;
	j						: INT;
	l						: INT;
///////////////////////////////////////////////////////////////////////
    FBChart : FB_Chart;  		(* Instance of the data capturing FB *)
    Distance : REAL;             (* Distance input value *)
    Force : REAL;                (* Force input value *)
  	Showgraphtg:R_TRIG;
	bshowgraph:BOOL;
	SID:INT:=1;
	Item:INT;
	bSumSID:BOOL; 
	bSubSID:BOOL;
	bSumSIDtg:R_TRIG; 
	bSubSIDtg:R_TRIG;
	bEndstorege:BOOL;
	Endstoragetg: R_TRIG;
	rtrigProcessdata:R_TRIG;
	stProccessReportLogKils				:ARRAY [1..1]OF ST_ProcessReport;
	idx1:INT; 
	idx2:INT;
	idx3:INT; 
	idx0: INT;
END_VAR

ACT_StatusBanner();
MapUnitEventsToHMI();
ACT_ScreensNamesSet();
ACT_Outputs();
ACT_UserConf();
ACT_Inputs();
ACT_ShutdownAndQuit();
ACT_StatisticsReset();
ACT_DataGraph();
ACT_KisltlerHMI();

ACTION ACT_DataGraph:

FbChart(
	StartSignal:= K_Master_Kistler.eState=E_KistlerState.PRESS_CYCLE , 
	EndSignal:=  K_Master_Kistler.eState=E_KistlerState.PRESS_READY , 
	DistanceInput:= K_Master_Kistler.rKistlerLive_X, 
	ForceInput:=  K_Master_Kistler.rKistlerLive_Y, 
	DatosOut=>  , 
	bFinished=> ,  );

//Show Graph 

Showgraphtg(CLK:=K_Master_Kistler.eState=E_KistlerState.PRESS_READY); 
(*
IF Showgraphtg.Q THEN
	bshowgraph:=TRUE; 
	ELSIF K_Master_Kistler.eState=E_KistlerState.PRESS_CYCLE THEN
		bshowgraph:=FALSE; 
END_IF
*)
// Control Chart History 
 
	bSumSIDtg(CLK:=bSumSID);
	bSubSIDtg(CLK:=bSubSID);

// Navegation Chart 	
IF bSumSIDtg.Q THEN 
	SID:=SID+1;

	bSumSID:=FALSE;
END_IF

IF bSubSIDtg.Q THEN 
	SID:=SID-1;

	bSubSID:=FALSE;
END_IF

IF SID >10 THEN
	SID:=1;
END_IF

IF SID < 1 THEN
	SID:=10;
END_IF


//Storage Chart History 
(*IF FbChart.bFinished THEN 
	FOR STOI := 1 TO 99 DO	
	GVL_PERSISTENT.GraphDataHistorystorage[GVL_PERSISTENT.h, STOI].x := FbChart.DatosOut[1, STOI].x;
	GVL_PERSISTENT.GraphDataHistorystorage[GVL_PERSISTENT.h, STOI].y := FbChart.DatosOut[1, STOI].y;
	bEndstorege:= TRUE; 
END_FOR
END_IF
*)
rtrigProcessdata(CLK:=C_Machine_CTRL.eCycleState=E_ProcessCycle.Saving_DATA);

IF rtrigProcessdata.Q THEN 
	
	FOR idx0:=1 TO 100 DO 
		GVL_HMI.Graphdata[1, idx0].x := 0;
		GVL_HMI.Graphdata[1, idx0].y := 0;
	END_FOR
	
	FOR idx1 := 10 TO 2 BY -1 DO
    FOR idx2 := 1 TO 99 DO
		GVL_PERSISTENT.GraphDataHistorystorage[idx1,idx2]:=GVL_PERSISTENT.GraphDataHistorystorage[idx1-1, idx2];
	END_FOR
	END_FOR
	
	FOR idx3 := 1 TO 99 DO	
	
	GVL_PERSISTENT.GraphDataHistorystorage[1, idx3].x := FbChart.DatosOut[1, idx3].x;
	GVL_PERSISTENT.GraphDataHistorystorage[1, idx3].y := FbChart.DatosOut[1, idx3].y;
	GVL_HMI.Graphdata[1, idx3].x := FbChart.DatosOut[1, idx3].x;
	GVL_HMI.Graphdata[1, idx3].y := FbChart.DatosOut[1, idx3].y;
	bEndstorege:= TRUE; 
	END_FOR

END_IF		

Endstoragetg(CLK:=bEndstorege );

IF Endstoragetg.Q THEN 
	GVL_PERSISTENT.h:=	GVL_PERSISTENT.h+1;
	bEndstorege:=FALSE;
END_IF

// Clean Chart
FOR Item := 1 TO 99 DO
	GVL_HMI.GraphDataHistory[1, Item].x := 0;
	GVL_HMI.GraphDataHistory[1, Item].y := 0;
END_FOR

// Load Chart according SID index  
FOR Item := 1 TO 99 DO
	GVL_HMI.GraphDataHistory[1, Item].x := GVL_PERSISTENT.GraphDataHistorystorage[SID, Item].x;
	GVL_HMI.GraphDataHistory[1, Item].y := GVL_PERSISTENT.GraphDataHistorystorage[SID, Item].y;
END_FOR

//Load Data in tab
stProccessReportLogKils[1]:= GVL_PERSISTENT.stProccessReportLog[SID];
END_ACTION

ACTION ACT_Inputs:
tonButtonPressed( IN :=	GVL_HMI.bSmacCyc1 				OR
						GVL_HMI.bSmacCyc2 				OR
						GVL_HMI.bY_AxisPosition1 		OR
						GVL_HMI.bY_AxisPosition2 		OR
						GVL_HMI.bY_AxisPosition3 		OR
						GVL_HMI.bY_HomePosition			OR
						GVL_HMI.bKistlerCycle			OR
						GVL_HMI.bSmacSetValue			OR
						GVL_HMI.bSmacHOME				OR
						GVL_HMI.bMoveToPos				OR
						GVL_HMI.bResetSmacGoodParts		OR
						GVL_HMI.bResetSmacBadParts		OR
						GVL_HMI.bResetKistlerGoodParts 	OR
						GVL_HMI.bResetKistlerBadParts	OR
						GVL_HMI.bQuitHmi				,
					PT := T#500MS);
					
IF 	tonButtonPressed.Q THEN
	GVL_HMI.bSmacCyc1 				:= FALSE;
	GVL_HMI.bSmacCyc2 				:= FALSE;
	GVL_HMI.bY_AxisPosition1		:= FALSE;
	GVL_HMI.bY_AxisPosition2 		:= FALSE;
	GVL_HMI.bY_AxisPosition3 		:= FALSE;
	GVL_HMI.bY_HomePosition			:= FALSE;
	GVL_HMI.bKistlerCycle			:= FALSE;
	GVL_HMI.bSmacSetValue			:= FALSE;
	GVL_HMI.bSmacHOME				:= FALSE;
	GVL_HMI.bMoveToPos				:= FALSE;
	GVL_HMI.bResetSmacGoodParts		:= FALSE;
	GVL_HMI.bResetSmacBadParts		:= FALSE;
	GVL_HMI.bResetKistlerGoodParts 	:= FALSE;
	GVL_HMI.bResetKistlerBadParts	:= FALSE;
	GVL_HMI.bQuitHmi				:= FALSE;
END_IF
END_ACTION

ACTION ACT_KisltlerHMI:
OpenKistlerHMI(
    NetId := '',
	PathStr := 'C:\Windows\System32\cmd.exe',
    DirName := 'C:\Windows\System32',
    ComndLine := '/c start "" "C:\Users\ADMINISTRATOR\Desktop\Kistler"',
    Start := GVL_HMI.bKistlerHMI,
    TmOut := DEFAULT_ADS_TIMEOUT
);
(*OpenKistlerHMI( too Slow
    NetId   := '',
    PathStr := 'C:\Windows\System32\WindowsPowerShell\v1.0\powershell.exe',
    DirName := 'C:\Windows\System32\WindowsPowerShell\v1.0',
    ComndLine := '-WindowStyle Hidden -Command "Start-Process" C:\Users\ADMINISTRATOR\Desktop\Kistler.lnk',
    Start   := GVL_HMI.bKistlerHMI,
    TmOut   := DEFAULT_ADS_TIMEOUT
);*)
 
GVL_HMI.bKistlerHMI:= FALSE;
END_ACTION

ACTION ACT_Outputs:
//SMAC
GVL_HMI.nCurrentDistanceSmac 	:= (stSmacIO.inCurrentValueLinear /200);

fbScaleSmacMan(	rRawData				:= stSmacIO.inCurrentPositionLinear,
				rRawDataLowerOffLimit	:= 0,
				rRawDataUpperOffLimit	:= S_Master_SMAC.I_O_fbSmacCycleMan.nScaledLinearSetPoint,
				rScaleDataLowerOffLimit	:= -141,
				rScaleDataUpperOffLimit	:= -58,
				rY_Intercept			:= -141,
				rScaleData				=> GVL_HMI.rSmacAnimationMan);
				
				
fbScaleKistlerMan(	rRawData				:= GVL_HMI.rKistlerLiveReading_X,
				rRawDataLowerOffLimit	:= 0,
				rRawDataUpperOffLimit	:= 28.6,
				rScaleDataLowerOffLimit	:= -120,
				rScaleDataUpperOffLimit	:= 0,
				rY_Intercept			:= -120,
				rScaleData				=> GVL_HMI.rKistlerAnimationMan);
				
				
fbScaleSmacCyc(	rRawData				:= stSmacIO.inCurrentPositionLinear,
				rRawDataLowerOffLimit	:= 0,
				rRawDataUpperOffLimit	:= S_Master_SMAC.I_O_fbSmacCycleMan.nScaledLinearSetPoint,
				rScaleDataLowerOffLimit	:= -110,
				rScaleDataUpperOffLimit	:= -10,
				rY_Intercept			:= -110,
				rScaleData				=> GVL_HMI.rSmacAnimationCyc);
				
				
fbScaleKistlerCyc(	rRawData				:= GVL_HMI.rKistlerLiveReading_X,
				rRawDataLowerOffLimit	:= 0,
				rRawDataUpperOffLimit	:= 30,
				rScaleDataLowerOffLimit	:= -80,
				rScaleDataUpperOffLimit	:= 50,
				rY_Intercept			:= -80,
				rScaleData				=> GVL_HMI.rKistlerAnimationCyc);

IF GVL_HMI.bScrewAnimation THEN
	fbScaleScrew(	rRawData				:= stSmacIO.inCurrentPositionLinear,
				rRawDataLowerOffLimit	:= 0,
				rRawDataUpperOffLimit	:= S_Master_SMAC.I_O_fbSmacCycleMan.nScaledLinearSetPoint,
				rScaleDataLowerOffLimit	:= 310,
				rScaleDataUpperOffLimit	:= 400,
				rY_Intercept			:= 330,
				rScaleData				=> GVL_HMI.rScrewAnimation);
				GVL_HMI.bScrewPartPresent:= TRUE;

ELSE 			GVL_HMI.rScrewAnimation	:= 400;
				GVL_HMI.bScrewPartPresent:= GVL_MASTER.bScrew_Present;
END_IF
			
	GVL_HMI.bLinearServoEnabled			:= GVL_MODULES.stSmacIO.inStatusWordLinear.1;
	GVL_HMI.bLinearHomingSuccess		:= GVL_MODULES.stSmacIO.inStatusWordLinear.6;
	GVL_HMI.bLinearPhasingSuccess		:= GVL_MODULES.stSmacIO.inStatusWordLinear.8;
	GVL_HMI.bLinearError				:= GVL_MODULES.stSmacIO.inStatusWordLinear.13;
	
	GVL_HMI.bRotativeServoEnabled		:= GVL_MODULES.stSmacIO.inStatusWordRotative.1;
	GVL_HMI.bRotativeHomingSuccess		:= GVL_MODULES.stSmacIO.inStatusWordRotative.6;
	GVL_HMI.bRotativePhasingSuccess		:= GVL_MODULES.stSmacIO.inStatusWordRotative.8;
	GVL_HMI.bRotativeError				:= GVL_MODULES.stSmacIO.inStatusWordRotative.13;
	
	GVL_HMI.bSmacSTO1Fault				:= (GVL_MODULES.stSmacIO.inStatusWordLinear.16 OR
											GVL_MODULES.stSmacIO.inStatusWordRotative.16);
	GVL_HMI.bSmacSTO2Fault				:= (GVL_MODULES.stSmacIO.inStatusWordLinear.17 OR
											GVL_MODULES.stSmacIO.inStatusWordRotative.17);
	GVL_HMI.bSmacGeneralFault			:= (GVL_MODULES.stSmacIO.inStatusWordLinear.12 OR
											GVL_MODULES.stSmacIO.inStatusWordRotative.12);
END_ACTION

ACTION ACT_ScreensNamesSet:
	
	GVL_HMI.aManualScreens[0]			:='SMAC / AXIS Y';
	GVL_HMI.aManualScreens[1]			:='KISTLER / AXIS Y';
	
	GVL_HMI.aSettingScreens[0]			:='KISTLER';
	GVL_HMI.aSettingScreens[1]			:='SMAC';
	GVL_HMI.aSettingScreens[2]			:='AXIS Y';
	
	
	GVL_HMI.aIOScreens[0]			:='Overview';
	GVL_HMI.aIOScreens[1]			:='HMI - CP2913-0000 | Beckhoff HMI';
	GVL_HMI.aIOScreens[2]			:='PLC - C6015-0010 | Beckhoff PLC | Windows 10 Embedded';
	GVL_HMI.aIOScreens[3]			:='Terminal 1- EK1100 | EtherCAT Coupler';
	GVL_HMI.aIOScreens[4]			:='Terminal 2 - EL6070 | Licence';
	GVL_HMI.aIOScreens[5]			:='Terminal 3 - EL6910 | Safe PLC';
	GVL_HMI.aIOScreens[6]			:='TERMINAL 4 _ EL1918 - 8 Channel Digital Safety Inputs';
	GVL_HMI.aIOScreens[7]			:='TERMINAL 5 _ EL1918 - 8 Channel Digital Safety Inputs';
	GVL_HMI.aIOScreens[8]			:='TERMINAL 6 _ ELEL2904 - 4 Channel Digital Safety Outputs';
	GVL_HMI.aIOScreens[9]			:='TERMINAL 7 _ ELEL2904 - 4 Channel Digital Safety Outputs';
	GVL_HMI.aIOScreens[10]			:='TERMINAL 8 _ EL1809 - 16 Channel Digital Input Terminal';
	GVL_HMI.aIOScreens[11]			:='TERMINAL 9 _ EL1809 - 16 Channel Digital Input Terminal';
	GVL_HMI.aIOScreens[12]			:='TERMINAL 10 _ EL2809	- 16 Channel Digital Output Terminal';
	GVL_HMI.aIOScreens[13]			:='TERMINAL 11 _ EL9576 - Brake Chopper Terminal';
	GVL_HMI.aIOScreens[14]			:='TERMINAL 12 _ EL7211-0010 - Servo Motor Drive';
	GVL_HMI.aIOScreens[15]			:='BOX 13 _ maXYnos - Drive and Force Sensor for Kistler Press';
	GVL_HMI.aIOScreens[16]			:='BOX 14 _ SMAC - Linear amd Rotative axis for screw part';
END_ACTION

ACTION ACT_ShutdownAndQuit:
closeChrome(
    NetId := '',
    PathStr := 'C:\Windows\System32\mshta vbscript:Execute("CreateObject(""WScript.Shell"").Run ""powershell -c',
    DirName := 'C:\Windows\System32\WindowsPowerShell\v1.0',
    ComndLine := 'taskkill /F /IM chrome.exe /T"", 0: window.close")',
    Start := GVL_HMI.bQuitHmi,
    TmOut := DEFAULT_ADS_TIMEOUT
);
 
GVL_HMI.bQuitHmi:= FALSE;

ntShutdown(NETID := GVL_HMI.ntAMSNetID, DELAY := 5, START := GVL_HMI.bShutDown);
END_ACTION

ACTION ACT_StatisticsReset:
IF GVL_HMI.bResetSmacGoodParts THEN
	GVL_PERSISTENT.nSmacGoodParts	:= 0;	
END_IF
IF GVL_HMI.bResetSmacBadParts THEN
	GVL_PERSISTENT.nSmacBadParts	:= 0;	
END_IF
IF GVL_HMI.bResetKistlerGoodParts THEN
	GVL_PERSISTENT.nKistlerGoodParts	:= 0;	
END_IF
IF GVL_HMI.bResetKistlerBadParts THEN
	GVL_PERSISTENT.nKistlerBadParts	:= 0;	
END_IF
END_ACTION

ACTION ACT_StatusBanner:
//Machine status banner action
//SYSTEM POWER UP
IF GVL_MASTER.stMachineStatus.bSystemPowerUp THEN	
	GVL_MASTER.stMachineStatus.sMachineStatusText := 'SYSTEM POWER UP';		// fill colour WHITE, text colour BLACK
	GVL_MASTER.stMachineStatus.nMachineStatusColour := nWHITE;
	GVL_MASTER.stMachineStatus.nMachineStatusTxtCol := nBLACK;
	GVL_MASTER.stMachineStatus.sBannerBckColor := sWHITE;
	GVL_MASTER.stMachineStatus.sBannerTextColor := sBLACK;
END_IF

(* IMMEDIATE STOPPED *)
IF GVL_MASTER.stMachineStatus.bImmediateStopped THEN	
	GVL_MASTER.stMachineStatus.sMachineStatusText := 'IMMEDIATE STOPPED';		// fill colour BLACK, text colour WHITE
	GVL_MASTER.stMachineStatus.nMachineStatusColour := nBLACK;
	GVL_MASTER.stMachineStatus.nMachineStatusTxtCol := nWHITE;
	GVL_MASTER.stMachineStatus.sBannerBckColor := sBLACK;
	GVL_MASTER.stMachineStatus.sBannerTextColor := sWHITE;	
END_IF

(* SYSTEM INITIALISING *)
IF GVL_MASTER.stMachineStatus.bInitialising THEN	
	GVL_MASTER.stMachineStatus.sMachineStatusText := 'SYSTEM INITIALIZING';		// fill colour YELLOW, text colour BLACK
	GVL_MASTER.stMachineStatus.nMachineStatusColour := nYELLOW;
	GVL_MASTER.stMachineStatus.nMachineStatusTxtCol := nBLACK;
	GVL_MASTER.stMachineStatus.sBannerBckColor := sYELLOW;
	GVL_MASTER.stMachineStatus.sBannerTextColor := sBLACK;
END_IF

(* SYSTEM READY TO START FLASH ON *)
IF GVL_MASTER.stMachineStatus.bReadyToStart AND GVL_UTILITIES.bFlash1Hz THEN
	GVL_MASTER.stMachineStatus.sMachineStatusText := 'SYSTEM READY TO START';		// fill colour GREEN, text colour WHITE
	GVL_MASTER.stMachineStatus.nMachineStatusColour := nGREEN;
	GVL_MASTER.stMachineStatus.nMachineStatusTxtCol := nWHITE;
	GVL_MASTER.stMachineStatus.sBannerBckColor := sGREEN;
	GVL_MASTER.stMachineStatus.sBannerTextColor := sWHITE;
END_IF

(* SYSTEM READY TO START FLASH OFF *)
IF GVL_MASTER.stMachineStatus.bReadyToStart AND NOT GVL_UTILITIES.bFlash1Hz THEN	
	GVL_MASTER.stMachineStatus.sMachineStatusText := 'SYSTEM READY TO START';		// fill colour WHITE, text colour GREEN
	GVL_MASTER.stMachineStatus.nMachineStatusColour := nWHITE;
	GVL_MASTER.stMachineStatus.nMachineStatusTxtCol := nGREEN;
	GVL_MASTER.stMachineStatus.sBannerBckColor := sWHITE;
	GVL_MASTER.stMachineStatus.sBannerTextColor := sGREEN;
END_IF

(* SYSTEM AUTO CYCLE *)
IF GVL_MASTER.stMachineStatus.bAutoCycle  THEN	
	GVL_MASTER.stMachineStatus.sMachineStatusText := 'SYSTEM AUTO CYCLE';		// fill colour GREEN, text colour WHITE
	GVL_MASTER.stMachineStatus.nMachineStatusColour := nGREEN;
	GVL_MASTER.stMachineStatus.nMachineStatusTxtCol := nWHITE;
	GVL_MASTER.stMachineStatus.sBannerBckColor := sGREEN;
	GVL_MASTER.stMachineStatus.sBannerTextColor := sWHITE;	
END_IF

(* STOPPING *)
IF GVL_MASTER.stMachineStatus.bStopping AND GVL_UTILITIES.bFlash1Hz THEN	
	GVL_MASTER.stMachineStatus.sMachineStatusText := 'STOPPING';		// fill colour BLACK, text colour WHITE
	GVL_MASTER.stMachineStatus.nMachineStatusColour := nBLACK;
	GVL_MASTER.stMachineStatus.nMachineStatusTxtCol := nWHITE;
	GVL_MASTER.stMachineStatus.sBannerBckColor := sBLACK;
	GVL_MASTER.stMachineStatus.sBannerTextColor := sWHITE;	
END_IF

(* STOPPING *)
IF GVL_MASTER.stMachineStatus.bStopping AND NOT GVL_UTILITIES.bFlash1Hz THEN	
	GVL_MASTER.stMachineStatus.sMachineStatusText := 'STOPPING';		// fill colour WHITE, text colour BLACK
	GVL_MASTER.stMachineStatus.nMachineStatusColour := nWHITE;
	GVL_MASTER.stMachineStatus.nMachineStatusTxtCol := nBLACK;
	GVL_MASTER.stMachineStatus.sBannerBckColor := sWHITE;
	GVL_MASTER.stMachineStatus.sBannerTextColor := sBLACK;	
END_IF

(* CYCLE STOPPED *)
IF GVL_MASTER.stMachineStatus.bCycleStopped THEN	
	GVL_MASTER.stMachineStatus.sMachineStatusText := 'CYCLE STOPPED';		// fill colour BLACK, text colour WHITE
	GVL_MASTER.stMachineStatus.nMachineStatusColour := nBLACK;
	GVL_MASTER.stMachineStatus.nMachineStatusTxtCol := nWHITE;
	GVL_MASTER.stMachineStatus.sBannerBckColor := sBLACK;
	GVL_MASTER.stMachineStatus.sBannerTextColor := sWHITE;	
END_IF

(* IMMEDIATE FAULT FLASH ON *)
IF GVL_MASTER.stMachineStatus.bImmediateFault AND GVL_UTILITIES.bFlash1Hz THEN	
	GVL_MASTER.stMachineStatus.sMachineStatusText := 'IMMEDIATE FAULT';		// fill colour RED, text colour WHITE
	GVL_MASTER.stMachineStatus.nMachineStatusColour := nRED;
	GVL_MASTER.stMachineStatus.nMachineStatusTxtCol := nWHITE;
	GVL_MASTER.stMachineStatus.sBannerBckColor := sRED;
	GVL_MASTER.stMachineStatus.sBannerTextColor := sWHITE;	
END_IF

(* IMMEDIATE FAULT FLASH OFF *)
IF GVL_MASTER.stMachineStatus.bImmediateFault AND NOT GVL_UTILITIES.bFlash1Hz THEN	
	GVL_MASTER.stMachineStatus.sMachineStatusText := 'IMMEDIATE FAULT';		// fill colour WHITE, text colour BLACK
	GVL_MASTER.stMachineStatus.nMachineStatusColour := nWHITE;
	GVL_MASTER.stMachineStatus.nMachineStatusTxtCol := nBLACK;
	GVL_MASTER.stMachineStatus.sBannerBckColor := sWHITE;
	GVL_MASTER.stMachineStatus.sBannerTextColor := sBLACK;	
END_IF

(* CYCLE STOP FAULT FLASH ON *)
IF GVL_MASTER.stMachineStatus.bCycleStopFault AND GVL_UTILITIES.bFlash1Hz THEN	
	GVL_MASTER.stMachineStatus.sMachineStatusText := 'CYCLE STOP FAULT';		// fill colour RED, text colour WHITE
	GVL_MASTER.stMachineStatus.nMachineStatusColour := nRED;
	GVL_MASTER.stMachineStatus.nMachineStatusTxtCol := nWHITE;
	GVL_MASTER.stMachineStatus.sBannerBckColor := sRED;
	GVL_MASTER.stMachineStatus.sBannerTextColor := sWHITE;	
END_IF

(* CYCLE STOP FAULT FLASH OFF *)
IF GVL_MASTER.stMachineStatus.bCycleStopFault AND NOT GVL_UTILITIES.bFlash1Hz THEN	
	GVL_MASTER.stMachineStatus.sMachineStatusText := 'CYCLE STOP FAULT';		// fill colour WHITE, text colour RED
	GVL_MASTER.stMachineStatus.nMachineStatusColour := nWHITE;
	GVL_MASTER.stMachineStatus.nMachineStatusTxtCol := nRED;
	GVL_MASTER.stMachineStatus.sBannerBckColor := sWHITE;
	GVL_MASTER.stMachineStatus.sBannerTextColor := sRED;	
END_IF

(* MANUAL MODE *)
IF GVL_MASTER.stMachineStatus.bManualMode THEN	
	GVL_MASTER.stMachineStatus.sMachineStatusText := 'MANUAL MODE';		// fill colour BLUE text colour WHITE
	GVL_MASTER.stMachineStatus.nMachineStatusColour := nBLUE;
	GVL_MASTER.stMachineStatus.nMachineStatusTxtCol := nWHITE;
	GVL_MASTER.stMachineStatus.sBannerBckColor := sBLUE;
	GVL_MASTER.stMachineStatus.sBannerTextColor := sWHITE;	
END_IF
END_ACTION

ACTION ACT_UserConf:
//Getting user group

Tc2_Utilities.DELETE2( ADR(GVL_HMI.sUserGroup), ADR(sUserGroupID), NSize, Nlen, nPos) ;

IF sUserGroupID = 'Administ' THEN
	
	GVL_HMI.sUserGroup2 := 'Administrator';//Final User String

ELSE GVL_HMI.sUserGroup2 := sUserGroupID;
	

END_IF
//Logout 

tonUserLogOut( IN := (sUserGroupID = 'Administ' OR sUserGroupID ='Engineer') AND GVL_HMI.bUserLogedIntSignal , PT := T#10M);

IF tonUserLogOut.Q AND (sUserGroupID = 'Administ' OR sUserGroupID ='Engineer') THEN
	
	GVL_HMI.bLogOut 	:= TRUE;

	ELSE GVL_HMI.bLogOut := FALSE;

END_IF

tUserLoggedIn( IN := GVL_HMI.bUserLogedIntSignal, PT := T#2S);

rUserLoggedIn( CLK := tUserLoggedIn.Q);

IF rUserLoggedIn.Q THEN
	bUserLoggedIn := TRUE;
END_IF

IF bUserLoggedIn THEN
	
	GVL_PERSISTENT.stUserLogHMI[GVL_PERSISTENT.UserId].UserLog := GVL_HMI.sUserName;
	GVL_PERSISTENT.stUserLogHMI[GVL_PERSISTENT.UserId].UserLogTime := GVL_MASTER.sSystemTime;
	GVL_PERSISTENT.stUserLogHMI[GVL_PERSISTENT.UserId].UserLogDate := GVL_MASTER.sSystemDate;
	GVL_PERSISTENT.UserId := GVL_PERSISTENT.UserId + 1;
	bUserLoggedIn := FALSE;

END_IF

IF GVL_PERSISTENT.stUserLogHMI[200].UserLog <> '' THEN
	
GVL_PERSISTENT.stUserLogHMI[0].UserLog 					:= GVL_PERSISTENT.stUserLogHMI[200].UserLog;
GVL_PERSISTENT.stUserLogHMI[0].UserLogTime				:= GVL_PERSISTENT.stUserLogHMI[200].UserLogTime;
GVL_PERSISTENT.stUserLogHMI[0].UserLogDate				:= GVL_PERSISTENT.stUserLogHMI[200].UserLogDate;
GVL_PERSISTENT.stUserLogHMI[200].UserLog 				:= '';
GVL_PERSISTENT.stUserLogHMI[200].UserLogTime 			:= '';
GVL_PERSISTENT.stUserLogHMI[200].UserLogDate			:= '';
GVL_PERSISTENT.UserId			:= 1;


END_IF
END_ACTION

METHOD MapUnitEventsToHMI : BOOL
VAR_INPUT
END_VAR
VAR
	i		:INT; 	//Unit index
	j		:INT;	//Unit event index
	k		:INT; 	//HMI event index	
END_VAR
//Set event texts first
IF GVL_Master.stAlarms[0].bEventTextsSet AND
   GVL_Master.stAlarms[1].bEventTextsSet AND
   GVL_Master.stAlarms[2].bEventTextsSet AND
   GVL_Master.stAlarms[3].bEventTextsSet AND
   NOT GVL_HMI.bEventTextsSet 
THEN
	SetEventTexts();
		
	GVL_HMI.bEventTextsSet := TRUE;
END_IF

//Map events from master and stations into HMI events
IF GVL_HMI.bEventTextsSet THEN
	k := 0; 
	FOR i := 0 TO 3 DO
		FOR j := 0 TO 128 - 1 DO
			GVL_HMI.aEventFlags[k] := GVL_Master.stAlarms[i].aEventFlags[j];
			k := k + 1;
		END_FOR
	END_FOR
END_IF
END_METHOD

METHOD SetEventTexts : BOOL
VAR_INPUT
END_VAR
VAR
	i				:INT; 	//Unit index
	j				:INT;	//HMI event index
	k				:INT;	//
END_VAR
//Set global event texts based on unit event texts (master and stations
k := 0;
FOR i := 0 TO 3 DO
	//For each unit (master, station1, station2)
	//Alarm texts
	FOR j := 0 TO 99 DO
		fbStringFormatter(	sFormat := 'Alarm No. %d - %s', 
					 	arg1 := F_INT(k), 
						arg2 := F_String(GVL_Master.stAlarms[i].aEventTexts[j]),
						sOut => GVL_HMI.aEventTexts[k]);
						
		k := k + 1; //Increment global events index
	END_FOR
	
	//Messages
	FOR j := 100 TO 127 DO
		fbStringFormatter(	sFormat := 'Message No. %d - %s', 
					 		arg1 := F_INT(k), 
							arg2 := F_String(GVL_Master.stAlarms[i].aEventTexts[j]),
							sOut => GVL_HMI.aEventTexts[k]);
							
		k := k + 1; //Increment global events index
	END_FOR
END_FOR
END_METHOD

END_PROGRAM

// ---- POUs/03_Utilities/FB_Scale.TcPOU
FUNCTION_BLOCK FB_Scale
VAR_INPUT
	rRawData                   	: LREAL;
	rRawDataLowerOffLimit      	: LREAL;
	rRawDataUpperOffLimit      	: LREAL;
	rScaleDataLowerOffLimit    	: LREAL;
	rScaleDataUpperOffLimit    	: LREAL;
	rY_Intercept				: LREAL;
	
END_VAR
VAR_OUTPUT
	rScaleData					: LREAL;
END_VAR
VAR
	m							: LREAL;
END_VAR

IF (rRawDataUpperOffLimit - rRawDataLowerOffLimit <> 0) THEN
	m								:= (rScaleDataUpperOffLimit - rScaleDataLowerOffLimit )/( rRawDataUpperOffLimit - rRawDataLowerOffLimit);

END_IF

rScaleData						:= ( rRawData * m) + rY_Intercept;

END_FUNCTION_BLOCK

// ---- POUs/03_Utilities/FB_Chart.TcPOU
FUNCTION_BLOCK FB_Chart
VAR_INPUT
    StartSignal : BOOL;           // Signal to start capturing data
    EndSignal   : BOOL;           // Signal to stop capturing data
    DistanceInput : REAL;         // Incoming distance value
    ForceInput    : REAL;         // Incoming force value
	h:INT;						  //Index History persitent
END_VAR

VAR_OUTPUT
    DatosOut : ARRAY[1..1,1..100] OF Stpoint;  // Output array with captured data
  	bFinished  : BOOL;                     // TRUE when finished
END_VAR

VAR
	IsCapturing : BOOL;                     // TRUE while capturing
    Timer : TON;                   // Internal timer
	d:INT;
    ind : INT := 1;              // Internal index (start from 1)
	Endcycletg : R_TRIG;
	
END_VAR

	Endcycletg(CLK:=EndSignal);
// Start the timer only when StartSignal is TRUE and EndSignal is FALSE
Timer(IN := IsCapturing, PT := T#40ms);

// Main logic


IF StartSignal (*AND NOT EndSignal*) THEN
	FOR D := 1 TO 100 DO
        DatosOut[1, d].x := 0.0;  // Poner la coordenada X a 0
        DatosOut[1, d].y := 0.0;  // Poner la coordenada Y a 0
    END_FOR
	
	ind:=1;
    IsCapturing := TRUE;
    bFinished := FALSE;
END_IF 

IF IsCapturing AND NOT EndSignal AND NOT StartSignal THEN
    IF Timer.Q AND ind <= 199 THEN
        // Store current values in the array
        DatosOut[1,ind].x := DistanceInput;
        DatosOut[1,ind].y := ForceInput;
	
        ind := ind + 1;

        // Reset the timer for the next 1-second interval
        Timer(IN := FALSE);  // Stop
        Timer(IN := TRUE);   // Restart
    END_IF


ELSIF Endcycletg.Q OR ind > 199 THEN
    // Stop capturing when signal is given or array is full
    IsCapturing := FALSE;
 
	ind:=1;
    // Stop the timer
    Timer(IN := FALSE);
END_IF

bFinished:=Endcycletg.Q;

END_FUNCTION_BLOCK

// ---- POUs/00_MASTER/D_FaultHandling.TcPOU
PROGRAM D_FaultHandling
VAR
	i							: INT;
	bFlagResetOn				: BOOL;
	bStationCycleFaultFlag		: BOOL;
END_VAR

ACT_FaultTrig();

(************************************** Faults reset **********************************************)
IF   bResetButtonRisingEdge THEN 
	FOR i := 0 TO 127 DO
		GVL_MASTER.stAlarms[0].aEventFlags[i] := FALSE;
	END_FOR
END_IF


//===============================================================
//Initialize event texts on first scan
IF NOT GVL_MASTER.stAlarms[0].bEventTextsSet THEN
	SetEventTexts();
	GVL_MASTER.stAlarms[0].bEventTextsSet := TRUE;
END_IF
IF NOT GVL_MASTER.stAlarms[0].bEventTextsSet THEN
	GVL_MASTER.stAlarms[0].bEventTextsSet := FALSE;
END_IF


(***************************************************************************************************)
//Immediate fault
GVL_MASTER.stAlarms[0].bImmediateFault := FALSE;
FOR i := 0 TO 32DO
	GVL_MASTER.stAlarms[0].bImmediateFault := GVL_MASTER.stAlarms[0].bImmediateFault OR GVL_MASTER.stAlarms[0].aEventFlags[i];
END_FOR

//Cycle stop fault
GVL_MASTER.stAlarms[0].bCycleStopFault := FALSE;
FOR i := 33 TO 79 DO
	GVL_MASTER.stAlarms[0].bCycleStopFault := GVL_MASTER.stAlarms[0].bCycleStopFault OR GVL_MASTER.stAlarms[0].aEventFlags[i];
END_FOR

//Cycle stop request
GVL_MASTER.stAlarms[0].bCycleStopRequest := FALSE;
FOR i := 80 TO 99 DO
	GVL_MASTER.stAlarms[0].bCycleStopRequest := GVL_MASTER.stAlarms[0].bCycleStopRequest OR GVL_MASTER.stAlarms[0].aEventFlags[i];
END_FOR


(**************************** Master Fault Monitors ***********************************************)
(* Station Immediate Fault Monitor *)
stMasterCTRL.bNoMachineImmediateFault	 := 	NOT GVL_MASTER.stAlarms[0].bImmediateFault AND NOT GVL_MASTER.stAlarms[1].bImmediateFault AND
                                            			NOT GVL_MASTER.stAlarms[2].bImmediateFault AND NOT GVL_MASTER.stAlarms[3].bImmediateFault;
								
(**************************************************************************************************)

(* Master Cycle Stop Fault Monitor *)
 stMasterCtrl.bNoCycleStopFault:= NOT GVL_MASTER.stAlarms[0].bCycleStopFault AND NOT GVL_MASTER.stAlarms[1].bCycleStopFault AND
								NOT GVL_MASTER.stAlarms[2].bCycleStopFault AND NOT GVL_MASTER.stAlarms[3].bCycleStopFault;
(* Cycle Stop Request *)
IF GVL_MASTER.stAlarms[0].bCycleStopRequest OR GVL_MASTER.stAlarms[1].bCycleStopRequest OR 
	GVL_MASTER.stAlarms[2].bCycleStopRequest OR GVL_MASTER.stAlarms[3].bCycleStopRequest THEN
	stMasterCtrl.bCycleStopRequest			:= TRUE;
ELSE stMasterCtrl.bCycleStopRequest			:= FALSE;
END_IF

ACTION ACT_FaultTrig:
(**************************************************************************************************)
(**************************** Master Immediate Fault Stop *****************************************)
(**************************************************************************************************)
//TERMINAL 1 _ EK1100 - EtherCAT Coupler Not Operational
IF NOT GVL_MASTER.stMachineStatus.bSystemPowerUp AND GVL_IO.nEK1100State<>8 THEN
	GVL_MASTER.stAlarms[0].aEventFlags[1] := TRUE;
END_IF
// TERMINAL 2 _ EL6070-0033	- License Key Terminal for TC3 Not Operational
IF NOT GVL_MASTER.stMachineStatus.bSystemPowerUp AND GVL_IO.nEL6070State<>8 THEN
	GVL_MASTER.stAlarms[0].aEventFlags[2] := TRUE;
END_IF
// TERMINAL 3 _ EL6910 - Safety PLC - Virtual Channels Not Operational
IF NOT GVL_MASTER.stMachineStatus.bSystemPowerUp AND GVL_IO.nEL6910State<>8 THEN
	GVL_MASTER.stAlarms[0].aEventFlags[3] := TRUE;
END_IF
// TERMINAL 4 _ EL1918 - 8 Channel Digital Safety Inputs Not Operational
IF NOT GVL_MASTER.stMachineStatus.bSystemPowerUp AND GVL_IO.nEL1918_1State<>8 THEN
	GVL_MASTER.stAlarms[0].aEventFlags[4] := TRUE;
END_IF
// TERMINAL 5 _ EL1918 - 8 Channel Digital Safety Inputs Not Operational
IF NOT GVL_MASTER.stMachineStatus.bSystemPowerUp AND GVL_IO.nEL1918_2State<>8 THEN
	GVL_MASTER.stAlarms[0].aEventFlags[5] := TRUE;
END_IF
// TERMINAL 6 _ ELEL2904 - 4 Channel Digital Safety Outputs Not Operational
IF NOT GVL_MASTER.stMachineStatus.bSystemPowerUp AND GVL_IO.nEL2904_1State<>8 THEN
	GVL_MASTER.stAlarms[0].aEventFlags[6] := TRUE;
END_IF
// TERMINAL 7 _ ELEL2904 - 4 Channel Digital Safety Outputs Not Operational
IF NOT GVL_MASTER.stMachineStatus.bSystemPowerUp AND GVL_IO.nEL2904_2State<>8 THEN
	GVL_MASTER.stAlarms[0].aEventFlags[7] := TRUE;
END_IF
// TERMINAL 8 _ EL1809 - 16 Channel Digital Input Terminal Not Operational
IF NOT GVL_MASTER.stMachineStatus.bSystemPowerUp AND GVL_IO.nEL1809_1State<>8 THEN
	GVL_MASTER.stAlarms[0].aEventFlags[8] := TRUE;
END_IF
// TERMINAL 9 _ EL1809 - 16 Channel Digital Input Terminal Not Operational
IF NOT GVL_MASTER.stMachineStatus.bSystemPowerUp AND GVL_IO.nEL1809_2State<>8 THEN
	GVL_MASTER.stAlarms[0].aEventFlags[9] := TRUE;
END_IF
// TERMINAL 10 _ EL2809	- 16 Channel Digital Output Terminal Not Operational
IF NOT GVL_MASTER.stMachineStatus.bSystemPowerUp AND GVL_IO.nEL2809State<>8 THEN
	GVL_MASTER.stAlarms[0].aEventFlags[10] := TRUE;
END_IF
// TERMINAL 11 _ EL9576 - Brake Chopper Terminal Not Operational
IF NOT GVL_MASTER.stMachineStatus.bSystemPowerUp AND GVL_IO.nEL9576State<>8 THEN
	GVL_MASTER.stAlarms[0].aEventFlags[11] := TRUE;
END_IF
// TERMINAL 12 _ EL7211-0010 - Servo Motor Drive Not Operational
IF NOT GVL_MASTER.stMachineStatus.bSystemPowerUp AND GVL_IO.nEL7211State<>8 THEN
	GVL_MASTER.stAlarms[0].aEventFlags[12] := TRUE;
END_IF
//No user logged in
GVL_MASTER.stAlarms[0].aEventTimers[13](IN := (GVL_HMI.sUserName=''), PT := T#40MS);
IF GVL_MASTER.stAlarms[0].aEventTimers[13].Q THEN
	GVL_MASTER.stAlarms[0].aEventFlags[13] := TRUE;	
END_IF
//Safety 
IF NOT stSafety.bSafety_OK THEN
	GVL_MASTER.stAlarms[0].aEventFlags[14] := TRUE;
END_IF
//E-STOP Pressed
IF NOT stSafety.bEStop_OK THEN
	GVL_MASTER.stAlarms[0].aEventFlags[15] := TRUE;
END_IF
//Light beam Crossed
IF NOT stSafety.bLightBeam_MuteCMD AND stSafety.bLightBeam_Crossed AND NOT Y_Master_Y_Axis.refY_Axis.Status.Moving THEN
	GVL_MASTER.stAlarms[0].aEventFlags[16] := TRUE;
END_IF
//Door openned
IF NOT stSafety.bDoorClosed AND stSafety.bLockDoor_CMD  THEN
	GVL_MASTER.stAlarms[0].aEventFlags[17] := TRUE;
END_IF
//PSU 1 FAULT
IF NOT GVL_IO.iPSU_1_OK  THEN
	GVL_MASTER.stAlarms[0].aEventFlags[18] := TRUE;
END_IF
//PSU 2 FAULT
IF NOT GVL_IO.iPSU_2_OK  THEN
	GVL_MASTER.stAlarms[0].aEventFlags[19] := TRUE;
END_IF
//PSU 3 FAULT
IF NOT GVL_IO.iPSU_3_OK  THEN
	GVL_MASTER.stAlarms[0].aEventFlags[20] := TRUE;
END_IF
//E-Stop CH1 Signal
IF NOT GVL_IO.iE_Stop_Ch1  THEN
	GVL_MASTER.stAlarms[0].aEventFlags[21] := TRUE;
END_IF
//E-Stop CH2 Signal
IF NOT GVL_IO.iE_Stop_Ch2  THEN
	GVL_MASTER.stAlarms[0].aEventFlags[22] := TRUE;
END_IF



//System stopping timeout
GVL_MASTER.stAlarms[0].aEventTimers[13](IN := ( GVL_MASTER.stMachineStatus.bStopping), PT := T#20S);
IF GVL_MASTER.stAlarms[0].aEventTimers[13].Q THEN
	GVL_MASTER.stAlarms[0].aEventFlags[13] := TRUE;	
END_IF
//10 Min Auto cycle stop
GVL_MASTER.stAlarms[0].aEventTimers[80](IN := ((C_Machine_CTRL.eCycleState = E_ProcessCycle.IDLE) AND 
(stMachineStatus.eMachineState = E_MachineState.SYSTEM_AUTO_CYCLE)), PT := T#10M);
IF GVL_MASTER.stAlarms[0].aEventTimers[80].Q THEN //
	GVL_MASTER.stAlarms[0].aEventFlags[80] := TRUE;
END_IF
//Autocyle Timeout 
(*GVL_MASTER.stAlarms[0].aEventTimers[81]
(IN:= GVL_MASTER.stMachineStatus.bAutoCycle AND C_Machine_CTRL.eCycleState <> E_ProcessCycle.IDLE , PT :=T#90S ); 
IF GVL_MASTER.stAlarms[0].aEventTimers[81].Q THEN
	GVL_MASTER.stAlarms[0].aEventFlags[81] := TRUE;
END_IF*)
//No user logged IN
IF NOT GVL_HMI.bUserLogedIntSignal THEN
	GVL_MASTER.stAlarms[0].aEventFlags[82] := TRUE;
END_IF
END_ACTION

METHOD SetEventTexts : BOOL
VAR_INPUT
END_VAR
//Immediate Faults
GVL_MASTER.stAlarms[0].aEventTexts[0] := '';
GVL_MASTER.stAlarms[0].aEventTexts[1] := 'TERMINAL 1 _ EK1100 - EtherCAT Coupler Not Operational';
GVL_MASTER.stAlarms[0].aEventTexts[2] := 'TERMINAL 2 _ EL6070-0033	- License Key Terminal for TC3 Not Operational';
GVL_MASTER.stAlarms[0].aEventTexts[3] := 'TERMINAL 3 _ EL6910 - Safety PLC - Virtual Channels Not Operational';
GVL_MASTER.stAlarms[0].aEventTexts[4] := 'TERMINAL 4 _ EL1918 - 8 Channel Digital Safety Inputs Not Operational';
GVL_MASTER.stAlarms[0].aEventTexts[5] := 'TERMINAL 5 _ EL1918 - 8 Channel Digital Safety Inputs Not Operational';
GVL_MASTER.stAlarms[0].aEventTexts[6] := 'TERMINAL 6 _ ELEL2904 - 4 Channel Digital Safety Outputs Not Operational';
GVL_MASTER.stAlarms[0].aEventTexts[7] := 'TERMINAL 7 _ ELEL2904 - 4 Channel Digital Safety Outputs Not Operational';
GVL_MASTER.stAlarms[0].aEventTexts[8] := 'TERMINAL 8 _ EL1809 - 16 Channel Digital Input Terminal Not Operational';
GVL_MASTER.stAlarms[0].aEventTexts[9] := 'TERMINAL 9 _ EL1809 - 16 Channel Digital Input Terminal Not Operational';
GVL_MASTER.stAlarms[0].aEventTexts[10] := 'TERMINAL 10 _ EL2809	- 16 Channel Digital Output Terminal Not Operational';
GVL_MASTER.stAlarms[0].aEventTexts[11] := 'TERMINAL 11 _ EL9576 - Brake Chopper Terminal Not Operational'; 
GVL_MASTER.stAlarms[0].aEventTexts[12] := 'TERMINAL 12 _ EL7211-0010 - Servo Motor Drive Not Operational';
GVL_MASTER.stAlarms[0].aEventTexts[13] := 'No user logged in';
GVL_MASTER.stAlarms[0].aEventTexts[14] := 'Safety';
GVL_MASTER.stAlarms[0].aEventTexts[15] := 'E-STOP Pressed';
GVL_MASTER.stAlarms[0].aEventTexts[16] := 'Light beam Crossed';
GVL_MASTER.stAlarms[0].aEventTexts[17] := 'Door openned';
GVL_MASTER.stAlarms[0].aEventTexts[18] := 'PSU 1 FAULT';
GVL_MASTER.stAlarms[0].aEventTexts[19] := 'PSU 2 FAULT';
GVL_MASTER.stAlarms[0].aEventTexts[20] := 'PSU 3 FAULT';
GVL_MASTER.stAlarms[0].aEventTexts[21] := 'E-Stop CH1 Signal';
GVL_MASTER.stAlarms[0].aEventTexts[22] := 'E-Stop CH2 Signal';

//Cycle stop fault

GVL_MASTER.stAlarms[0].aEventTexts[33] := 'System stopping timeout';
GVL_MASTER.stAlarms[0].aEventTexts[34] := '10 Min Auto cycle stop';
GVL_MASTER.stAlarms[0].aEventTexts[35] := 'Autocyle Timeout';
GVL_MASTER.stAlarms[0].aEventTexts[36] := '';
GVL_MASTER.stAlarms[0].aEventTexts[37] := '';
GVL_MASTER.stAlarms[0].aEventTexts[38] := '';
GVL_MASTER.stAlarms[0].aEventTexts[39] := '';
GVL_MASTER.stAlarms[0].aEventTexts[40] := ''; 
GVL_MASTER.stAlarms[0].aEventTexts[41] := '';
GVL_MASTER.stAlarms[0].aEventTexts[42] := '';
GVL_MASTER.stAlarms[0].aEventTexts[43] := '';
GVL_MASTER.stAlarms[0].aEventTexts[44] := '';
GVL_MASTER.stAlarms[0].aEventTexts[45] := '';
GVL_MASTER.stAlarms[0].aEventTexts[46] := '';
GVL_MASTER.stAlarms[0].aEventTexts[47] := '';
GVL_MASTER.stAlarms[0].aEventTexts[48] := '';
GVL_MASTER.stAlarms[0].aEventTexts[59] := '';
GVL_MASTER.stAlarms[0].aEventTexts[50] := '';

//Cycle Stop Requests

GVL_MASTER.stAlarms[0].aEventTexts[80] := '10 Min Auto cycle stop';
GVL_MASTER.stAlarms[0].aEventTexts[81] := 'Autocyle Timeout';
GVL_MASTER.stAlarms[0].aEventTexts[82] := 'No user logged IN';

GVL_MASTER.stAlarms[0].aEventTexts[84] := '';
GVL_MASTER.stAlarms[0].aEventTexts[85] := '';
GVL_MASTER.stAlarms[0].aEventTexts[86] := '';
GVL_MASTER.stAlarms[0].aEventTexts[87] := ''; 
GVL_MASTER.stAlarms[0].aEventTexts[88] := '';
GVL_MASTER.stAlarms[0].aEventTexts[89] := '';
END_METHOD

END_PROGRAM

// ---- POUs/03_Utilities/PRG_SysPulses.TcPOU
PROGRAM PRG_SysPulses
VAR 
// 50% Duty Cycle
	fbXO_250Hz    		:FB_Pulse;	//Correct at 2ms tick
	fbXO_50Hz     		:FB_Pulse;	//Correct at 2ms tick
	fbXO_10Hz			:FB_Pulse;	//Correct at 2ms tick
	fbXO_5Hz			:FB_Pulse;	//Correct at 2ms tick
	fbXO_2Hz			:FB_Pulse;	//Correct at 2ms tick	
	fbXO_1Hz			:FB_Pulse;	//Correct at 2ms tick
	fbXO_05Hz			:FB_Pulse;	//Correct at 2ms tick
	// Frictions
	fbXO_1p85Hz			:FB_Pulse;	//Correct at 2ms tick
	fbXO_1p52Hz			:FB_Pulse;	//Correct at 2ms tick
	fbXO_1p33Hz			:FB_Pulse;	//Correct at 2ms tick
	fbXO_1p19Hz			:FB_Pulse;	//Correct at 2ms tick	
	
// 70/30 Duty Cycle
	fbXO_1Hz_7030		:FB_Pulse;	//Correct at 2ms tick
	
// 80/20 Duty Cycle
	fbXO_1Hz_8020		:FB_Pulse;	//Correct at 2ms tick
//-----------------------------------------------oldschoo1		
END_VAR

(*** Oscilator Pulse Generators at 2ms tick ***)

// 50% Duty Cycle
	fbXO_250Hz(
		bEnable				:=	TRUE,
		tPulseOn			:=	T#2MS,
		tPulseOff			:=	T#2MS,
		bFlash				=>	bFlash250Hz);
	fbXO_50Hz( 
		bEnable	    		:=	TRUE,
		tPulseOn			:=	T#10MS,
		tPulseOff			:=	T#10MS,
		bFlash				=>	bFlash50Hz);
	fbXO_10Hz(
		bEnable				:=	TRUE,
		tPulseOn			:=	T#50MS,
		tPulseOff			:=	T#50MS,
		bFlash				=>	bFlash10Hz);
	fbXO_5Hz(
		bEnable				:=	TRUE,
		tPulseOn			:=	T#100MS,
		tPulseOff			:=	T#100MS,
		bFlash				=>	bFlash5Hz);
	fbXO_2Hz(
		bEnable				:=	TRUE,
		tPulseOn			:=	T#250MS,
		tPulseOff			:=	T#250MS,
		bFlash				=>	bFlash2Hz);
	fbXO_1Hz(
		bEnable				:=	TRUE,
		tPulseOn			:=	T#500MS,
		tPulseOff			:=	T#500MS,
		bFlash				=>	bFlash1Hz);	
	fbXO_05Hz(
		bEnable				:=	TRUE,
		tPulseOn			:=	T#1000MS,
		tPulseOff			:=	T#1000MS,
		bFlash				=>	bFlash05Hz);
//Frictions
	fbXO_1p85Hz(
		bEnable				:=	TRUE,
		tPulseOn			:=	T#270MS,
		tPulseOff			:=	T#270MS,
		bFlash				=>	bFlash1p85Hz);
	fbXO_1p52Hz(
		bEnable				:=	TRUE,
		tPulseOn			:=	T#330MS,
		tPulseOff			:=	T#330MS,
		bFlash				=>	bFlash1p52Hz);
	fbXO_1p33Hz(
		bEnable				:=	TRUE,
		tPulseOn			:=	T#376MS,
		tPulseOff			:=	T#376MS,
		bFlash				=>	bFlash1p33Hz);
	fbXO_1p19Hz(
		bEnable				:=	TRUE,
		tPulseOn			:=	T#416MS,
		tPulseOff			:=	T#416MS,
		bFlash				=>	bFlash1p2Hz);
		
// 70/30 Duty Cycle
	fbXO_1Hz_7030(
		bEnable				:=	TRUE,
		tPulseOn			:=	T#700MS,
		tPulseOff			:=	T#300MS,
		bFlash				=>	bFlash1Hz_7030);
		
// 80/20 Duty Cycle
	fbXO_1Hz_8020(
		bEnable				:=	TRUE,
		tPulseOn			:=	T#800MS,
		tPulseOff			:=	T#200MS,
		bFlash				=>	bFlash1Hz_8020);
//-----------------------------------------------oldschoo1

END_PROGRAM

// ---- POUs/03_Utilities/FB_Pulse.TcPOU
FUNCTION_BLOCK FB_Pulse
VAR_INPUT
	bEnable		    :BOOL;
	tPulseOn		:TIME;
	tPulseOff		:TIME;
//------------------------------------*
END_VAR
VAR
	tonXO_On		:Tc2_Standard.TON;
	tonXO_Off	    :Tc2_Standard.TON;
//------------------------------------*
END_VAR
VAR_OUTPUT
	bFlash			:BOOL;
//----------------------------oldschoo1	
END_VAR

// Enable
IF 	(bEnable AND NOT tonXO_Off.Q)		
	THEN
	tonXO_On.IN			:=TRUE;
ELSE
	tonXO_On.IN			:=FALSE;
END_IF

// Generate Pulse
tonXO_On(
	IN:= ,
	PT:= tPulseOff,
	Q=> ,
	ET=>
	);
tonXO_Off(
	IN:= tonXO_On.Q,
	PT:= tPulseOn,
	Q=> ,
	ET=>
	);
	
// Oscilator Output
bFlash	:=	tonXO_On.Q;
//-------------------------------oldschoo1

END_FUNCTION_BLOCK

// ---- POUs/03_Utilities/FB_TerminalInfo.TcPOU
FUNCTION_BLOCK FB_TerminalInfo
VAR_INPUT
	nTerminalState  : UINT;
END_VAR
VAR_OUTPUT
	sTerminalState  : STRING;
END_VAR
VAR
END_VAR

IF nTerminalState = 1 THEN 
   sTerminalState := 'Initialization';
ELSIF  nTerminalState = 2 THEN 
   sTerminalState := 'PREOP';  
ELSIF  nTerminalState = 3 THEN 
   sTerminalState := 'BOOT'; 
ELSIF  nTerminalState = 4 THEN 
   sTerminalState := 'SAFEOP';   
ELSIF  nTerminalState = 8 THEN 
   sTerminalState := 'OPERATIONAL';
ELSIF  nTerminalState = 16#0010 THEN 
   sTerminalState := 'Slave signals error';   
ELSIF  nTerminalState = 16#0020 THEN 
   sTerminalState := 'Invalid vendorId, productCode... read';  
ELSIF  nTerminalState = 16#0040 THEN 
   sTerminalState := 'Initialization error occurred';   
ELSIF  nTerminalState = 16#0080 THEN 
   sTerminalState := 'Slave disabled';   
ELSIF  nTerminalState = 16#0100 THEN 
   sTerminalState := 'Slave not present';    
ELSIF  nTerminalState = 16#0200 THEN 
   sTerminalState := 'Slave signals link error';    
ELSIF  nTerminalState = 16#0400 THEN 
   sTerminalState := 'Slave signals missing link'; 
ELSIF  nTerminalState = 16#0800 THEN 
   sTerminalState := 'Slave signals unexpected link';
ELSIF  nTerminalState = 16#1000 THEN 
   sTerminalState := 'Communication port A';
ELSIF  nTerminalState = 16#2000 THEN 
   sTerminalState := 'Communication port B';
ELSIF  nTerminalState = 16#4000 THEN 
   sTerminalState := 'Communication port C';
ELSIF  nTerminalState = 16#8000 THEN 
   sTerminalState := 'Communication port D'; 	
END_IF

END_FUNCTION_BLOCK

// ---- POUs/01_MODULES/AXIS_Y/PRG_Fault_Axis_Y.TcPOU
PROGRAM PRG_Fault_Axis_Y
VAR
	i					: INT;
	bTest				: BOOL;
END_VAR
VAR_IN_OUT
  aAlarms  : ARRAY[0..3] OF ST_Events;
END_VAR

ACT_FaultTrig();

(************************************** Faults reset **********************************************)
IF   bResetButtonRisingEdge THEN 
	FOR i := 0 TO 127 DO
		GVL_MASTER.stAlarms[1].aEventFlags[i] := FALSE;
	END_FOR
END_IF
//===============================================================
//Initialize event texts on first scan
IF NOT GVL_MASTER.stAlarms[1].bEventTextsSet THEN
	SetEventTexts();
	GVL_MASTER.stAlarms[1].bEventTextsSet := TRUE;
END_IF


(***************************************************************************************************)
//Immediate fault
GVL_MASTER.stAlarms[1].bImmediateFault := FALSE;
FOR i := 0 TO 32DO
	GVL_MASTER.stAlarms[1].bImmediateFault := GVL_MASTER.stAlarms[1].bImmediateFault OR GVL_MASTER.stAlarms[1].aEventFlags[i];
END_FOR

//Cycle stop fault
GVL_MASTER.stAlarms[1].bCycleStopFault := FALSE;
FOR i := 33 TO 79 DO
	GVL_MASTER.stAlarms[1].bCycleStopFault := GVL_MASTER.stAlarms[1].bCycleStopFault OR GVL_MASTER.stAlarms[1].aEventFlags[i];
END_FOR

//Cycle stop REQUEST
GVL_MASTER.stAlarms[1].bCycleStopRequest := FALSE;
FOR i := 80 TO 99 DO
	GVL_MASTER.stAlarms[1].bCycleStopRequest := GVL_MASTER.stAlarms[1].bCycleStopRequest OR GVL_MASTER.stAlarms[1].aEventFlags[i];
END_FOR

ACTION ACT_FaultTrig:
//AXIS Y General Fault
IF (Y_Master_Y_Axis.refY_Axis.NcToPlc.ErrorCode <> 0) THEN
	GVL_MASTER.stAlarms[1].aEventFlags[1] := TRUE;
END_IF


//Station 1 - Axis Y Homing Time Out
GVL_MASTER.stAlarms[1].aEventTimers[80]
(IN := ((stMachineStatus.eMachineState = E_MachineState.SYSTEM_INITIALISING) AND 
NOT (Y_Master_Y_Axis.eState = E_AxisState.AXIS_READY)),PT:= T#30S );
IF GVL_MASTER.stAlarms[1].aEventTimers[80].Q  THEN 
	GVL_MASTER.stAlarms[1].aEventFlags[80] := TRUE;
END_IF

//Station 1 - Axis Y Out of limit
IF NOT (Y_Master_Y_Axis.posTarget > Y_Master_Y_Axis.fPositionLimitMin) OR
	NOT (Y_Master_Y_Axis.posTarget < Y_Master_Y_Axis.fPositionLimitMax) THEN 
	//GVL_MASTER.stAlarms[1].aEventFlags[81] := TRUE;
	//bTest									:= TRUE;
END_IF
END_ACTION

METHOD SetEventTexts : BOOL
VAR_INPUT
END_VAR
//Immediate Faults
GVL_MASTER.stAlarms[1].aEventTexts[1] := 'AXIS Y General Fault					';
GVL_MASTER.stAlarms[1].aEventTexts[2] := '';
GVL_MASTER.stAlarms[1].aEventTexts[3] := '';
GVL_MASTER.stAlarms[1].aEventTexts[4] := '';
GVL_MASTER.stAlarms[1].aEventTexts[5] := '';
GVL_MASTER.stAlarms[1].aEventTexts[6] := '';
GVL_MASTER.stAlarms[1].aEventTexts[7] := '';
GVL_MASTER.stAlarms[1].aEventTexts[8] := '';
GVL_MASTER.stAlarms[1].aEventTexts[9] := '';
GVL_MASTER.stAlarms[1].aEventTexts[10] := ''; 
GVL_MASTER.stAlarms[1].aEventTexts[11] := ''; 
GVL_MASTER.stAlarms[1].aEventTexts[12] := '';
GVL_MASTER.stAlarms[1].aEventTexts[13] := '';
GVL_MASTER.stAlarms[1].aEventTexts[14] := '';
GVL_MASTER.stAlarms[1].aEventTexts[15] := '';
GVL_MASTER.stAlarms[1].aEventTexts[16] := '';
GVL_MASTER.stAlarms[1].aEventTexts[17] := '';
GVL_MASTER.stAlarms[1].aEventTexts[18] := '';
GVL_MASTER.stAlarms[1].aEventTexts[19] := '';
GVL_MASTER.stAlarms[1].aEventTexts[20] := '';
GVL_MASTER.stAlarms[1].aEventTexts[21] := '';
GVL_MASTER.stAlarms[1].aEventTexts[22] := '';
GVL_MASTER.stAlarms[1].aEventTexts[23] := '';
GVL_MASTER.stAlarms[1].aEventTexts[24] := '';
GVL_MASTER.stAlarms[1].aEventTexts[25] := '';
GVL_MASTER.stAlarms[1].aEventTexts[36] := '';

//Cycle Stop Requests

GVL_MASTER.stAlarms[1].aEventTexts[80] := 'Station 1 - Axis Y Homing Time Out';
GVL_MASTER.stAlarms[1].aEventTexts[81] := 'Station 1 - Axis Y Out of limit';
GVL_MASTER.stAlarms[1].aEventTexts[82] := '';

GVL_MASTER.stAlarms[1].aEventTexts[84] := '';
GVL_MASTER.stAlarms[1].aEventTexts[85] := '';
GVL_MASTER.stAlarms[1].aEventTexts[86] := '';
GVL_MASTER.stAlarms[1].aEventTexts[87] := ''; 
GVL_MASTER.stAlarms[1].aEventTexts[88] := '';
GVL_MASTER.stAlarms[1].aEventTexts[89] := '';
END_METHOD

END_PROGRAM

// ---- POUs/01_MODULES/KISTLER/PRG_Fault_Kistler.TcPOU
PROGRAM PRG_Fault_Kistler
VAR
	i					: INT;
	bTest				: BOOL;
END_VAR
VAR_IN_OUT
  aAlarms  : ARRAY[0..3] OF ST_Events;
END_VAR

ACT_FaultTrig();

(************************************** Faults reset **********************************************)
IF   bResetButtonRisingEdge THEN 
	FOR i := 0 TO 127 DO
		GVL_MASTER.stAlarms[2].aEventFlags[i] := FALSE;
	END_FOR
END_IF
//===============================================================
//Initialize event texts on first scan
IF NOT GVL_MASTER.stAlarms[2].bEventTextsSet THEN
	SetEventTexts();
	GVL_MASTER.stAlarms[2].bEventTextsSet := TRUE;
END_IF


(***************************************************************************************************)
//Immediate fault
GVL_MASTER.stAlarms[2].bImmediateFault := FALSE;
FOR i := 0 TO 32DO
	GVL_MASTER.stAlarms[2].bImmediateFault := GVL_MASTER.stAlarms[2].bImmediateFault OR GVL_MASTER.stAlarms[2].aEventFlags[i];
END_FOR

//Cycle stop fault
GVL_MASTER.stAlarms[2].bCycleStopFault := FALSE;
FOR i := 33 TO 79 DO
	GVL_MASTER.stAlarms[2].bCycleStopFault := GVL_MASTER.stAlarms[2].bCycleStopFault OR GVL_MASTER.stAlarms[2].aEventFlags[i];
END_FOR

//Cycle stop REQUEST
GVL_MASTER.stAlarms[2].bCycleStopRequest := FALSE;
FOR i := 80 TO 99 DO
	GVL_MASTER.stAlarms[2].bCycleStopRequest := GVL_MASTER.stAlarms[2].bCycleStopRequest OR GVL_MASTER.stAlarms[2].aEventFlags[i];
END_FOR

ACTION ACT_FaultTrig:
//Station 2 - Kistler Alarm
GVL_MASTER.stAlarms[2].aEventTimers[1]
(IN := K_Master_Kistler.stReceived.bAlarm AND NOT stMachineStatus.bImmediateFault AND NOT stMachineStatus.bInitialising , PT := T#500MS);
IF  GVL_MASTER.stAlarms[2].aEventTimers[1].Q THEN 
	GVL_MASTER.stAlarms[2].aEventFlags[1] := TRUE;
	bTest	:= TRUE;
END_IF
//Station 2 - Kistler Warning
GVL_MASTER.stAlarms[2].aEventTimers[2]
(IN := K_Master_Kistler.stReceived.bWarning AND NOT stMachineStatus.bImmediateFault AND NOT stMachineStatus.bInitialising , PT := T#500MS);
IF GVL_MASTER.stAlarms[2].aEventTimers[2].Q THEN 
	GVL_MASTER.stAlarms[2].aEventFlags[2] := TRUE;
	bTest := TRUE;
END_IF

//Station 2 - Kistler Homing Time Out
GVL_MASTER.stAlarms[2].aEventTimers[3]
(IN := (K_Master_Kistler.eState = E_KistlerState.GOTO_HOME_POS),PT:= T#30S );
IF GVL_MASTER.stAlarms[2].aEventTimers[80].Q  THEN 
	GVL_MASTER.stAlarms[2].aEventFlags[80] := TRUE;
END_IF
END_ACTION

METHOD SetEventTexts : BOOL
VAR_INPUT
END_VAR
//Immediate Faults
GVL_MASTER.stAlarms[2].aEventTexts[1] := 'Station 2 - Kistler Alarm';
GVL_MASTER.stAlarms[2].aEventTexts[2] := 'Station 2 - Kistler Warning';
GVL_MASTER.stAlarms[2].aEventTexts[3] := 'Station 2 - Kistler Homing Time Out';
GVL_MASTER.stAlarms[2].aEventTexts[4] := '';
GVL_MASTER.stAlarms[2].aEventTexts[5] := '';
GVL_MASTER.stAlarms[2].aEventTexts[6] := '';
GVL_MASTER.stAlarms[2].aEventTexts[7] := '';
GVL_MASTER.stAlarms[2].aEventTexts[8] := '';
GVL_MASTER.stAlarms[2].aEventTexts[9] := ''; 
GVL_MASTER.stAlarms[2].aEventTexts[10] := ''; 
GVL_MASTER.stAlarms[2].aEventTexts[11] := '';
GVL_MASTER.stAlarms[2].aEventTexts[12] := '';
GVL_MASTER.stAlarms[2].aEventTexts[13] := '';
GVL_MASTER.stAlarms[2].aEventTexts[14] := '';
GVL_MASTER.stAlarms[2].aEventTexts[15] := '';
GVL_MASTER.stAlarms[2].aEventTexts[16] := '';
GVL_MASTER.stAlarms[2].aEventTexts[17] := '';
GVL_MASTER.stAlarms[2].aEventTexts[18] := '';
GVL_MASTER.stAlarms[2].aEventTexts[19] := '';
GVL_MASTER.stAlarms[2].aEventTexts[20] := '';
GVL_MASTER.stAlarms[2].aEventTexts[21] := '';
GVL_MASTER.stAlarms[2].aEventTexts[22] := '';
GVL_MASTER.stAlarms[2].aEventTexts[28] := '';
GVL_MASTER.stAlarms[2].aEventTexts[29] := '';
GVL_MASTER.stAlarms[2].aEventTexts[30] := '';

//Cycle Stop Requests

GVL_MASTER.stAlarms[2].aEventTexts[80] := '';
GVL_MASTER.stAlarms[2].aEventTexts[81] := '';
GVL_MASTER.stAlarms[2].aEventTexts[82] := '';
GVL_MASTER.stAlarms[2].aEventTexts[84] := '';
GVL_MASTER.stAlarms[2].aEventTexts[85] := '';
GVL_MASTER.stAlarms[2].aEventTexts[86] := '';
GVL_MASTER.stAlarms[2].aEventTexts[87] := ''; 
GVL_MASTER.stAlarms[2].aEventTexts[88] := '';
GVL_MASTER.stAlarms[2].aEventTexts[89] := '';
END_METHOD

END_PROGRAM

// ---- POUs/03_Utilities/PRG_SysTime.TcPOU
PROGRAM PRG_SysTime
VAR
	//Variables
	bFirstRun						:BOOL:= TRUE;
	bReadyToRead					:BOOL;

	bUpdateSysTime					:BOOL; //Output of pulse generator
	tSysTimeUpdatePeriod			:TIME := T#5S;
	stTimeStamp						:TIMESTRUCT;
	stNullTimeStamp					:TIMESTRUCT;
	sRawDateTime					:STRING;
	sSystemDate						:STRING;
	sSystemTime						:STRING;
	sDateTime						:STRING;

	
	//Functions
	fbGetSystemTime					:TC2_Utilities.NT_GetTime;
	fbRTClock						:TC2_Utilities.RTC_EX2;		//Local real-time clock
	tonTimeUpdateGen				:TC2_Utilities.TON;			//Pulse generator for triggering fbGetSystemTime function
	rtrigSysTimeCollected			:TC2_Utilities.R_TRIG;		//System time collected

END_VAR
VAR_OUTPUT
		sDateTimeFormat				:STRING[40];
END_VAR

//Aux functions call
tonTimeUpdateGen(	IN := NOT bUpdateSysTime,
					PT := tSysTimeUpdatePeriod,
					Q => bUpdateSysTime);

//Get Current System Time
fbGetSystemTime(NETID := ,
				START := bFirstRun OR bUpdateSysTime,
				TMOUT := ,
				BUSY => ,
				ERR => ,
				ERRID => ,
				TIMESTR => );
				
//Get system time done detection - one-shot
rtrigSysTimeCollected(CLK := NOT fbGetSystemTime.BUSY);

//Synchronize Real-Time clock with system time
fbRTClock(	EN := rtrigSysTimeCollected.Q, 
			PDT := fbGetSystemTime.TIMESTR,
			CDT => stTimeStamp, 
			Q => bReadyToRead);

// System Date and Time in Proper Order 
IF bReadyToRead THEN
	sRawDateTime := SYSTEMTIME_TO_STRING(stTimeStamp);  // format: YYYY-MM-DD-hh:mm:ss.xxx
	sSystemDate := CONCAT(CONCAT(CONCAT(CONCAT(MID(sRawDateTime, 2, 9), '.'),  MID(sRawDateTime, 2, 6)), '.'), LEFT(sRawDateTime, 4));
	sSystemTime := MID(sRawDateTime, 8, 12);
	sDateTime := CONCAT(CONCAT(sSystemDate, '  '), sSystemTime);
	sDateTimeFormat	:= CONCAT(sDateTime, '    ');
END_IF;

bFirstRun := FALSE;

//by unknown dev

END_PROGRAM
